// TwinCAT 3 PLC project OC_Core
// Title: OC_Core
// Company: Open Commissioning
// Author: SpiraTec AG
// ProjectVersion: 1.3.1
// Description: Open Commissioning TwinCAT Core Library
// ProgramVersion: 3.1.4026.11
// libraries:
//   Tc2_Math, * (Beckhoff Automation GmbH)
//   Tc2_Standard, * (Beckhoff Automation GmbH)
//   Tc2_System, * (Beckhoff Automation GmbH)
//   Tc2_Utilities, * (Beckhoff Automation GmbH)
//   Tc3_Module, * (Beckhoff Automation GmbH)
//   TcUnit, * (www.tcunit.org)
// project tree:
//   Common/AdsMessageHandler/ FB_AdsMessageHandler.TcPOU, ST_AdsMessage.TcDUT
//   Common/Components/Encoder/ FB_Encoder.TcPOU, ST_Encoder_Config.TcDUT
//   Common/Components/ FB_DriveControl.TcPOU, FB_Clock.TcPOU, FB_ClockAdvanced.TcPOU, FB_Heater.TcPOU, FB_MoveAbsolute.TcPOU, FB_MoveVelocity.TcPOU, FB_Ping.TcPOU
//   Common/FileIo/ E_FileIoState.TcDUT, FB_FileIO.TcPOU
//   Common/Links/ FB_LinkDataReal.TcPOU, FB_LinkDevice.TcPOU, FB_LinkDataWord.TcPOU, FB_LinkDataLWord.TcPOU, FB_LinkDataDWord.TcPOU, FB_LinkDataByte.TcPOU
//   Common/RecordData/ FB_RecordData.TcPOU, I_RecordData.TcIO, ST_RecordIdent.TcDUT
//   Common/System/ E_ControllerType.TcDUT, FB_Base.TcPOU, FB_System.TcPOU, F_LogError.TcPOU, F_LogMessage.TcPOU, F_LogWarning.TcPOU, F_IsSystemValid.TcPOU, GVL_Core.TcGVL
//   Common/Utils/ E_NetworkByteOrder.TcDUT, F_Clamp01.TcPOU, F_GetHByte.TcPOU, F_Compare.TcPOU, F_GetLByte.TcPOU, F_Memcpy.TcPOU, F_Norm.TcPOU, F_ScaleLREAL.TcPOU, F_Sign.TcPOU, F_InverBytesOrder.TcPOU, ST_ScaleConfig.TcDUT
//   Devices/Basic/ FB_Device.TcPOU, FB_Panel.TcPOU, FB_Lock.TcPOU, FB_Cylinder.TcPOU, FB_DeviceByte.TcPOU, FB_DeviceLWord.TcPOU, FB_DeviceWord.TcPOU, FB_DeviceDWord.TcPOU, FB_DeviceReal.TcPOU, FB_Drive.TcPOU, FB_Button.TcPOU, FB_Lamp.TcPOU, FB_Reader.TcPOU, FB_Robot.TcPOU, FB_SensorAnalog.TcPOU, FB_SensorBinary.TcPOU, FB_Switch.TcPOU
//   / PlcTask.TcTTO
//   Tests/Common/ FB_AdsMessageHandler_Test.TcPOU, FB_Encoder_Test.TcPOU, FB_Memcpy_Test.TcPOU, FB_RecordData_Test.TcPOU, FB_Clamp01_Test.TcPOU, FB_Compare_Test.TcPOU, FB_InverBytesOrder_Test.TcPOU, FB_Norm_Test.TcPOU, FB_Sign_Test.TcPOU, FB_Scale_Test.TcPOU, FB_GetByte_Test.TcPOU, FB_System_Test.TcPOU
//   Tests/Components/ FB_DriveControl_Test.TcPOU, FB_Heater_Test.TcPOU, FB_MoveAbsolute_Test.TcPOU, FB_MoveVelocity_Test.TcPOU
//   Tests/Devices/ FB_Button_Test.TcPOU, FB_Device_Test.TcPOU, FB_Switch_Test.TcPOU, FB_Lock_Test.TcPOU, FB_DeviceReal_Test.TcPOU, FB_Panel_Test.TcPOU, FB_Robot_Test.TcPOU, FB_SensorBinary_Test.TcPOU, FB_SensorAnalog_Test.TcPOU, FB_Reader_Test.TcPOU, FB_Lamp_Test.TcPOU, FB_Cylinder_Test.TcPOU, FB_DeviceByte_Test.TcPOU, FB_Drive_Test.TcPOU, FB_DeviceLWord_Test.TcPOU, FB_DeviceWord_Test.TcPOU, FB_DeviceDWord_Test.TcPOU
//   Tests/ PRG_TEST.TcPOU

CONFIGURATION OC_Core
    RESOURCE PLC ON TwinCAT3
        TASK PlcTask(INTERVAL := T#1ms, PRIORITY := 1);
        PROGRAM PRG_TEST WITH PlcTask : PRG_TEST;
    END_RESOURCE
END_CONFIGURATION

// ---- Common/AdsMessageHandler/ST_AdsMessage.TcDUT
TYPE ST_AdsMessage :
STRUCT
	tNetID			: T_AmsNetID; // AMS NetId identifier
	tPort			: T_AmsPort; // AMS port number
	nInvokeID		: UDINT; // Unique identifier for the ADS invocation
	nIdxGrp			: UDINT; // Index group for the ADS command
	nIdxOffs		: UDINT; // Index offset within the ADS command
	nLength			: UDINT; // Length of the ADS message data
	nResult			: UDINT; // Result code from the ADS operation
	aData			: ARRAY[0..239] OF BYTE; // Data payload (240-byte buffer)
END_STRUCT
END_TYPE

// ---- Common/Components/Encoder/ST_Encoder_Config.TcDUT
TYPE ST_Encoder_Config :
STRUCT
	bIsIntegrator   		: BOOL := FALSE;  //Integrate input value
	fNumerator 	  			: REAL := 0.0001; //[unit/INC]
	fDenominator  			: REAL := 1.0; 	// Scaling
	fModulo 	  			: REAL := 0; // Modulo [unit]; If 0, will be ignored
	fGearFactor  			: REAL := 1.0;
	bInvertEncoderDirection : BOOL;
END_STRUCT
END_TYPE

// ---- Common/FileIo/E_FileIoState.TcDUT
{attribute 'conditionalshow'}
TYPE E_FileIoState :
(
	READY := 0,
	OPEN,
	CREATE,
	READ,
	WRITE,
	CLOSE,
	ERROR
);
END_TYPE

// ---- Common/RecordData/ST_RecordIdent.TcDUT
TYPE ST_RecordIdent :
STRUCT
	nPort  			: T_AmsPort; //ADS-Port of the Profinet Device. Ignored when using PLCSIM Advanced
	nSlot			: UINT; //Slotnumber of the Profinet Device. Ignored when using PLCSIM Advanced
	nSubSlot		: UINT; //Subslotnumber of the Profinet Device. Ignored when using PLCSIM Advanced
	nPlcId			: UINT; //Identifier of the PLC when using PLCSIM Advanced
	nHardwareId		: UINT; //Hardware-ID of the device when using PLCSIM Advanced
END_STRUCT
END_TYPE

// ---- Common/System/E_ControllerType.TcDUT
{attribute 'qualified_only'}
{attribute 'strict'}
TYPE E_ControllerType :
(
	NotDefined := 0,
	PlcSimAdvanced := 1
);
END_TYPE

// ---- Common/Utils/E_NetworkByteOrder.TcDUT
{attribute 'qualified_only'}
{attribute 'strict'}
TYPE E_NetworkByteOrder :
(
	BigEndian := 0, //Big Endian (MOTOROLA)
	LittleEndian := 1 //Little Endian (Intel)	
);
END_TYPE

// ---- Common/Utils/ST_ScaleConfig.TcDUT
{attribute 'pack_mode' := '0'} 
TYPE ST_ScaleConfig :
STRUCT
	fInputMin 	: LREAL := 0;
	fInputMax 	: LREAL := 100;
	fOutputMin 	: LREAL := 0;
	fOutputMax 	: LREAL := 65535;
END_STRUCT
END_TYPE

// ---- Common/System/GVL_Core.TcGVL
{attribute 'qualified_only'}
{attribute 'conditionalshow'}
VAR_GLOBAL	
	refSystem 			: REFERENCE TO FB_System;		
END_VAR

// ---- Common/RecordData/I_RecordData.TcIO
{attribute 'conditionalshow'}
INTERFACE I_RecordData

(*Send ADS Read Response message*)
METHOD SendReadResponse : HRESULT
VAR_INPUT
	stAdsMessage : ST_AdsMessage; //Response ADS Message
END_VAR
END_METHOD

(*Send ADS Write Response message*)
METHOD SendWriteResponse : HRESULT
VAR_INPUT
	stAdsMessage : ST_AdsMessage; //Response ADS Message
END_VAR
END_METHOD

(*Try to get a valid ADR read message. If the message is valid, the data in the input structure will be overwritten*)
METHOD GetReadIndication : BOOL
VAR_INPUT
	refDeviceAdsMessage : REFERENCE TO ST_AdsMessage; //Reference ADS Message
END_VAR
END_METHOD

(*Subscribe the RecordIdent device to the RecordData services. The RecordIdent device is initialised during subscription*)
METHOD Subscribe
VAR_INPUT
	pRecordIdent	: POINTER TO ST_RecordIdent; //Pointet to RecordIdent Device
	stAdsMessage 	: REFERENCE TO ST_AdsMessage; //Reference to the initial ADS message configuration of the device
END_VAR
END_METHOD

(*Try to get a valid ADR write message. If the message is valid, the data in the input structure will be overwritten*)
METHOD GetWriteIndication : BOOL
VAR_INPUT
	refDeviceAdsMessage : REFERENCE TO ST_AdsMessage; //Reference ADS Message
END_VAR
END_METHOD

END_INTERFACE

// ---- Tests/PRG_TEST.TcPOU
PROGRAM PRG_TEST
VAR
	FB_System_Test : FB_System_Test;
	FB_Clamp01_Test : FB_Clamp01_Test;
	FB_Compare_Test : FB_Compare_Test;
	FB_Norm_Test : FB_Norm_Test;
	FB_Scale_Test : FB_Scale_Test;
	FB_Sign_Test : FB_Sign_Test;
	FB_InverBytesOrder_Test : FB_InverBytesOrder_Test;
	FB_GetByte_Test : FB_GetByte_Test;
	FB_MEMCPY_Test : FB_MEMCPY_Test;
	FB_Heater_Test : FB_Heater_Test;
	FB_MoveVelocity_Test : FB_MoveVelocity_Test;
	FB_MoveAbsolute_Test : FB_MoveAbsolute_Test; 
	FB_DriveControl_Test : FB_DriveControl_Test;
	FB_Button_Test : FB_Button_Test;
	FB_Switch_Test : FB_Switch_Test;
	FB_Lock_Test : FB_Lock_Test;
	FB_Panel_Test : FB_Panel_Test;
	FB_Cylinder_Test : FB_Cylinder_Test;
	FB_Device_Test : FB_Device_Test;
	FB_DeviceByte_Test : FB_DeviceByte_Test;
	FB_DeviceWord_Test : FB_DeviceWord_Test;
	FB_DeviceDWord_Test : FB_DeviceDWord_Test;
	FB_DeviceLWord_Test : FB_DeviceLWord_Test;
	FB_DeviceReal_Test : FB_DeviceReal_Test;
	FB_Drive_Test : FB_Drive_Test;
	FB_Lamp_Test : FB_Lamp_Test;
	FB_Reader_Test : FB_Reader_Test;
	FB_SensorAnalog_Test : FB_SensorAnalog_Test;
	FB_SensorBinary_Test : FB_SensorBinary_Test;
	FB_Robot_Test : FB_Robot_Test;	
	FB_AdsMessageHandler_Test : FB_AdsMessageHandler_Test;
	FB_RecordData_Test : FB_RecordData_Test;
	FB_Encoder_Test : FB_Encoder_Test;	
END_VAR

TcUnit.RUN();

END_PROGRAM

// ---- Tests/Common/FB_System_Test.TcPOU
FUNCTION_BLOCK FB_System_Test EXTENDS TcUnit.FB_TestSuite
VAR
	_fbSystem : FB_System;
END_VAR

TestInitialization();
TestProperties();

METHOD TestInitialization
VAR
	fbGetCurTaskIdx 	: TC2_SYSTEM.GETCURTASKINDEX;
	fResult 	: REAL;
	fExpected 	: REAL;
	bResult 	: BOOL;
	bExpected 	: BOOL;
END_VAR
TEST('Before InitRun fTimeScaling is 0');
fExpected := 0;
fResult := _fbSystem.fTimeScaling;
AssertEquals(Expected := fExpected,
             Actual := fResult,
             Message := 'Result value is not correct');
TEST_FINISHED();

TEST('Before InitRun fDeltaTime is 0');
fExpected := 0;
fResult := _fbSystem.fDeltaTime;
AssertEquals(Expected := fExpected,
             Actual := fResult,
             Message := 'Result value is not correct');	
TEST_FINISHED();

TEST('Before InitRun GVL_IOSEF.refSystem is NULL');
bExpected := FALSE;
bResult := __ISVALIDREF(GVL_Core.refSystem);
AssertEquals(Expected := bExpected,
             Actual := bResult,
             Message := 'Result value is not correct');	
TEST_FINISHED();

_fbSystem();

TEST('After InitRun fTimeScaling > 0');
fExpected := 1;
fResult := _fbSystem.fTimeScaling;
AssertEquals(Expected := fExpected,
             Actual := fResult,
             Message := 'Result value is not correct');
TEST_FINISHED();

TEST('After InitRun fDeltaTime > 0');
fbGetCurTaskIdx();
fExpected := UDINT_TO_REAL(TwinCAT_SystemInfoVarList._TaskInfo[fbGetCurTaskIdx.index].CycleTime / 10000) / 1000.0;
fResult := _fbSystem.fDeltaTime;
AssertEquals(Expected := fExpected,
             Actual := fResult,
             Message := 'Result value is not correct');	
TEST_FINISHED();

TEST('After InitRun GVL_IOSEF.refSystem is Valid');
bExpected := TRUE;
bResult := __ISVALIDREF(GVL_Core.refSystem);
AssertEquals(Expected := bExpected,
             Actual := bResult,
             Message := 'Result value is not correct');	
TEST_FINISHED();
END_METHOD

METHOD TestProperties : REFERENCE TO FB_Test
VAR
	fbGetCurTaskIdx 	: TC2_SYSTEM.GETCURTASKINDEX;
	fResult 	: REAL;
	fExpected 	: REAL;
END_VAR
TEST('Test Property: bDebug');
_fbSystem.bDebug := TRUE;
AssertTRUE(Condition := _fbSystem.bDebug,  Message := 'Property value is not correct');	
TEST_FINISHED();

TEST('Test Property: bVerbose');
_fbSystem.bVerbose := TRUE;
AssertTRUE(Condition := _fbSystem.bVerbose,  Message := 'Property value is not correct');	
TEST_FINISHED();

TEST('Test Property: fTimeScaling Initial');
fExpected := 1;
fResult := _fbSystem.fTimeScaling;
AssertEquals(Expected := fExpected,
             Actual := fResult,
             Message := 'Result value is not correct');
TEST_FINISHED();

TEST('Test Property: fTimeScaling Zero');
_fbSystem.fTimeScaling := 0;
fExpected := 1;
fResult := _fbSystem.fTimeScaling;
AssertEquals(Expected := fExpected,
             Actual := fResult,
             Message := 'Result value is not correct');
TEST_FINISHED();

TEST('Test Property: fTimeScaling Limit Min');
_fbSystem.fTimeScaling := -1;
fExpected := 0.01000001;
fResult := _fbSystem.fTimeScaling;
AssertEquals(Expected := fExpected,
             Actual := fResult,
             Message := 'Result value is not correct');
TEST_FINISHED();

TEST('Test Property: fTimeScaling Limit Max');
_fbSystem.fTimeScaling := 1E+6;
fExpected := 100;
fResult := _fbSystem.fTimeScaling;
AssertEquals(Expected := fExpected,
             Actual := fResult,
             Message := 'Result value is not correct');
TEST_FINISHED();

TEST('Test Property: fTimeScaling In Range_1');
_fbSystem.fTimeScaling := 2;
fExpected := 2;
fResult := _fbSystem.fTimeScaling;
AssertEquals(Expected := fExpected,
             Actual := fResult,
             Message := 'Result value is not correct');
TEST_FINISHED();

TEST('Test Property: fTimeScaling In Range_2');
_fbSystem.fTimeScaling := 1;
fExpected := 1;
fResult := _fbSystem.fTimeScaling;
AssertEquals(Expected := fExpected,
             Actual := fResult,
             Message := 'Result value is not correct');
TEST_FINISHED();
END_METHOD

END_FUNCTION_BLOCK

// ---- Common/System/FB_System.TcPOU
(*
	FB_System should be defined and called up once in the project so that the GVL reference is correctly assigned. 
	If FB_System is not defined or there are several instances, the TwinCAT PLC project is forced into config mode with corresponding messages in the console.
*)
{attribute 'reflection'} 
FUNCTION_BLOCK FB_System
VAR_INPUT
	fbAdsMessageHandler 	: FB_AdsMessageHandler;
	fbRecordData 			: FB_RecordData(refAdsMessageHandler := fbAdsMessageHandler);
END_VAR

VAR
	{attribute 'simulation_interface'}
	Control				AT %Q* : BYTE;
	{attribute 'simulation_interface'}
	Status				AT %I* : BYTE;
	{attribute 'simulation_interface'}
	TimeScaling			AT %I* : REAL := 1.0;
	
	{attribute 'instance-path'} 
    {attribute 'noinit'} 
	_sPath 				: STRING;
	
	_bDebug				: BOOL;
	_bVerbose			: BOOL;
	_fDeltaTime 		: REAL;
	_fTimeScaling 		: REAL;
	_eControllerType	: E_ControllerType;
	
	_fbPing				: FB_Ping;
	
	{attribute 'hide'}
	_fbGetCurTaskIdx 	: TC2_SYSTEM.GETCURTASKINDEX;
END_VAR

InitRun();
fTimeScaling := TimeScaling;
_fbPing(bFeedback := Status.7, bTrigger => Control.7);

fbRecordData(); //Execution order -1 relative to FB_AdsMessageHandler
fbAdsMessageHandler();

PROPERTY bDebug : BOOL
GET
bDebug := _bDebug;
END_GET
SET
_bDebug := bDebug;
END_SET
END_PROPERTY

PROPERTY bVerbose : BOOL
GET
bVerbose := _bVerbose;
END_GET
SET
_bVerbose := bVerbose;
END_SET
END_PROPERTY

PROPERTY eControllerType : E_ControllerType
GET
eControllerType := _eControllerType;
END_GET
SET
_eControllerType := eControllerType;
END_SET
END_PROPERTY

PROPERTY PUBLIC fDeltaTime : REAL
GET
fDeltaTime := _fDeltaTime;
END_GET
SET // PRIVATE
_fDeltaTime := fDeltaTime;
END_SET
END_PROPERTY

PROPERTY PUBLIC fTimeScaling : REAL
GET
fTimeScaling := _fTimeScaling;
END_GET
SET
IF fTimeScaling = 0 THEN
	_fTimeScaling := 1.0;
ELSE
	_fTimeScaling := LIMIT(0.01000001, fTimeScaling, 100.0);	
END_IF
END_SET
END_PROPERTY

METHOD PRIVATE InitRun
VAR_INST
	bInitRun 			: BOOL := TRUE;
	sMessageFormat   	: T_MAXSTRING := '%s %s';
	sMessage  			: T_MAXSTRING;
	fbFormatString 		: FB_FormatString;
END_VAR
IF NOT bInitRun THEN RETURN; END_IF
bInitRun := FALSE;

IF __ISVALIDREF(GVL_Core.refSystem) THEN	
	fbFormatString(sFormat := sMessageFormat, arg1 := F_STRINGEx(_sPath), arg2 := F_STRINGEx('FB_System has no single instance! Check the PROGRAM declaration'), sOut => sMessage);
	ADSLOGSTR(msgCtrlMask := ADSLOG_MSGTYPE_ERROR, '%s', sMessage);	
ELSE 
	GVL_Core.refSystem REF= THIS^;
END_IF

_fbGetCurTaskIdx();
_fDeltaTime := UDINT_TO_REAL(TwinCAT_SystemInfoVarList._TaskInfo[_fbGetCurTaskIdx.index].CycleTime / 10000) / 1000.0;
_fTimeScaling := 1;

fbRecordData.eControllerType := _eControllerType;
END_METHOD

END_FUNCTION_BLOCK

// ---- Common/AdsMessageHandler/FB_AdsMessageHandler.TcPOU
(*ADS Message Handler is responsible for indication of the ADS Read/Write messages for local NetId and generation of the response message*)
FUNCTION_BLOCK FB_AdsMessageHandler
VAR_INPUT
	bDisable 				: BOOL;	//Deactivate cyclical execution
	bLog					: BOOL;	//Log ADS messages data in the console
	bVerbose				: BOOL; //Log Verbose information in the console
END_VAR

VAR	
	_fbAdsWriteIndicator 	: AdsWriteInd;	
	_fbAdsReadIndicator 	: AdsReadInd;
	_fbAdsWriteResponse		: AdsWriteRes;
	_fbAdsReadResponse		: AdsReadRes;	
	_stAdsMessageWrite		: ST_AdsMessage;
	_stAdsMessageRead		: ST_AdsMessage;
END_VAR

VAR CONSTANT
	S_FORMAT_RECEIVEWRITE	: STRING := 'AdsWriteInd Port: %X, IdxGrp: %X, IdxOffs: %X, InvokeId %X, Length: %X';
	S_FORMAT_RECEIVEREAD	: STRING := 'AdsReadInd Port: %X, IdxGrp: %X, IdxOffs: %X, InvokeId %X, Length: %X';
	S_FORMAT_RESPONSEWRITE	: STRING := 'AdsWriteRes Port: %X, IdxGrp: %X, IdxOffs: %X, InvokeId %X, Length: %X';
	S_FORMAT_RESPONSEREAD	: STRING := 'AdsReadRes Port: %X, IdxGrp: %X, IdxOffs: %X, InvokeId %X, Length: %X';  
END_VAR

IF bDisable THEN RETURN; END_IF

//Reset Indication and Result FBs
_fbAdsWriteResponse(RESPOND := FALSE);
_fbAdsReadResponse(RESPOND := FALSE);

//Capture all Write requests
_fbAdsWriteIndicator();
CreateAdsWriteMessage();
		
//Capture all Read requests
_fbAdsReadIndicator();
CreateAdsReadMessage();

(*Returns the status of the indication of the read message in the current frame*)
PROPERTY PUBLIC bIsAdsMessageReadValid : BOOL
GET
bIsAdsMessageReadValid := _stAdsMessageRead.tPort <> 0;
END_GET
END_PROPERTY

(*Returns the status of the indication of the write message in the current frame*)
PROPERTY PUBLIC bIsAdsMessageWriteValid : BOOL
GET
bIsAdsMessageWriteValid := _stAdsMessageWrite.tPort <> 0;
END_GET
END_PROPERTY

METHOD PRIVATE CreateAdsReadMessage : BOOL
IF NOT _fbAdsReadIndicator.VALID THEN RETURN; END_IF

MEMSET(ADR(_stAdsMessageRead), 0, SIZEOF(ST_AdsMessage));
_stAdsMessageRead.tNetId 		:= _fbAdsReadIndicator.NETID;
_stAdsMessageRead.tPort 		:= _fbAdsReadIndicator.PORT;
_stAdsMessageRead.nInvokeId 	:= _fbAdsReadIndicator.INVOKEID;
_stAdsMessageRead.nIdxGrp 		:= _fbAdsReadIndicator.IDXGRP;
_stAdsMessageRead.nIdxOffs 		:= _fbAdsReadIndicator.IDXOFFS;
_stAdsMessageRead.nLength 		:= _fbAdsReadIndicator.LENGTH;

IF bVerbose THEN
	LogAdsMessage(_stAdsMessageWrite, S_FORMAT_RECEIVEREAD);
END_IF

_fbAdsReadIndicator(CLEAR := TRUE);
_fbAdsReadIndicator(CLEAR := FALSE);
END_METHOD

METHOD PRIVATE CreateAdsWriteMessage : BOOL
IF NOT _fbAdsWriteIndicator.VALID THEN RETURN; END_IF

MEMSET(ADR(_stAdsMessageWrite), 0, SIZEOF(ST_AdsMessage));
_stAdsMessageWrite.tNetId 		:= _fbAdsWriteIndicator.NETID;
_stAdsMessageWrite.tPort 		:= _fbAdsWriteIndicator.PORT;
_stAdsMessageWrite.nInvokeId 	:= _fbAdsWriteIndicator.INVOKEID;
_stAdsMessageWrite.nIdxGrp 		:= _fbAdsWriteIndicator.IDXGRP;
_stAdsMessageWrite.nIdxOffs 	:= _fbAdsWriteIndicator.IDXOFFS;
_stAdsMessageWrite.nLength 		:= _fbAdsWriteIndicator.LENGTH;
			
//Limit size to 240
IF _stAdsMessageWrite.nLength > 240 THEN
	IF bVerbose THEN
		F_LOGWARNING(CONCAT('WRREC data length limited to 240. Requested data length was ', TO_STRING(_stAdsMessageWrite.nLength)));
	END_IF
	_stAdsMessageWrite.nLength := 240;
END_IF

MEMCPY(ADR(_stAdsMessageWrite.aData), _fbAdsWriteIndicator.DATAADDR, _stAdsMessageWrite.nLength);

IF bVerbose THEN
	LogAdsMessage(_stAdsMessageWrite, S_FORMAT_RECEIVEWRITE);
END_IF

_fbAdsWriteIndicator(CLEAR := TRUE);
_fbAdsWriteIndicator(CLEAR := FALSE);
END_METHOD

METHOD PRIVATE LogAdsMessage : BOOL
VAR_INPUT
	stAdsMessage 			: ST_AdsMessage;
	sFormat 				: STRING;
END_VAR

VAR
	fbFormatString			: FB_FormatString2;
	sMessage				: STRING;
END_VAR
fbFormatString(
	pFormatString := ADR(sFormat),
	arg1 := F_UINT(stAdsMessage.tPort),
	arg2 := F_UDINT(stAdsMessage.nIdxGrp),
	arg3 := F_UDINT(stAdsMessage.nIdxOffs),		
	arg4 := F_UDINT(stAdsMessage.nInvokeID),
	arg5 := F_UDINT(stAdsMessage.nLength),
	pDstString := ADR(sMessage),
	nDstSize := SIZEOF(sMessage));
F_LogMessage(sMessage);
END_METHOD

(*Send ADS Read Response message*)
METHOD PUBLIC SendReadResponse : HRESULT
VAR_INPUT
	stAdsMessage 	: ST_AdsMessage; //Response ADS Message
END_VAR
IF _fbAdsReadResponse.RESPOND THEN
	SendReadResponse := S_PENDING;
	RETURN;
END_IF

//Limit size to 240
IF stAdsMessage.nLength > 240 THEN
	IF bVerbose THEN
		F_LOGWARNING(CONCAT('RDRES data length limited to 240. Requested data length was ', TO_STRING(stAdsMessage.nLength)));
	END_IF
	stAdsMessage.nLength := 240;
END_IF

_fbAdsReadResponse(
	NETID:= stAdsMessage.tNetId, 
	PORT:= stAdsMessage.tPort, 
	INVOKEID:= stAdsMessage.nInvokeId, 
	RESULT:= stAdsMessage.nResult, 
	LEN:= stAdsMessage.nLength,
	DATAADDR:= ADR(stAdsMessage.aData),
	RESPOND:= TRUE);
IF bVerbose OR bLog THEN	
	LogAdsMessage(stAdsMessage, S_FORMAT_RESPONSEREAD);
END_IF

SendReadResponse := S_OK;
END_METHOD

(*Send ADS Write Response message*)
METHOD PUBLIC SendWriteResponse : HRESULT
VAR_INPUT
	stAdsMessage 	: ST_AdsMessage; //Response ADS Message
END_VAR
IF _fbAdsWriteResponse.RESPOND THEN
	SendWriteResponse := S_PENDING;
	RETURN;
END_IF

_fbAdsWriteResponse(
	NETID:= stAdsMessage.tNetId, 
	PORT:= stAdsMessage.tPort, 
	INVOKEID:= stAdsMessage.nInvokeId, 
	RESULT:= stAdsMessage.nResult, 
	RESPOND:= TRUE);	

IF bVerbose OR bLog THEN		
	LogAdsMessage(stAdsMessage, S_FORMAT_RESPONSEWRITE);
END_IF
	
SendWriteResponse := S_OK;
END_METHOD

(*Get last valid ADS Read Message*)
PROPERTY stAdsMessageRead : REFERENCE TO ST_AdsMessage
GET
stAdsMessageRead REF= _stAdsMessageRead;
END_GET
END_PROPERTY

(*Get last valid ADS Write Message*)
PROPERTY stAdsMessageWrite : REFERENCE TO ST_AdsMessage
GET
stAdsMessageWrite REF= _stAdsMessageWrite;
END_GET
END_PROPERTY

END_FUNCTION_BLOCK

// ---- Common/System/F_LogWarning.TcPOU
(*
	Log Warning message to TwinCAT console
*)
{attribute 'hide_all_locals'}
FUNCTION F_LogWarning : BOOL
VAR_INPUT
	sMessage : T_MAXSTRING;
END_VAR

VAR CONSTANT	
	S_LOGHEADER		: T_MAXSTRING := 'Open Commissioning: %s';
END_VAR

ADSLOGSTR(ADSLOG_MSGTYPE_WARN, S_LOGHEADER, sMessage);

END_FUNCTION

// ---- Common/System/F_LogMessage.TcPOU
(*
	Log message to TwinCAT console
*)
{attribute 'hide_all_locals'}
FUNCTION F_LogMessage : BOOL
VAR_INPUT
	sMessage : T_MAXSTRING;
END_VAR

VAR CONSTANT	
	S_LOGHEADER		: T_MAXSTRING := 'Open Commissioning: %s';
END_VAR

ADSLOGSTR(ADSLOG_MSGTYPE_HINT, S_LOGHEADER, sMessage);

END_FUNCTION

// ---- Common/RecordData/FB_RecordData.TcPOU
(*
	Uses an external ADS message handler (FB_AdsMessageHandler) for sending/receiving ADS messages.
	Handles cyclic execution for processing ADS messages and maintains a list of subscribed devices.	
*)
{attribute 'conditionalshow_all_locals}
FUNCTION_BLOCK PUBLIC FB_RecordData IMPLEMENTS I_RecordData
VAR_INPUT
	bDisable 				: BOOL; //Disables cyclic execution when set to TRUE
	bVerbose 				: BOOL; //Enables console logging of ADS message data
	eControllerType 		: E_ControllerType; //Determines data processing logic based on the controller type
END_VAR

VAR	
	_refAdsMessageHandler	: REFERENCE TO FB_AdsMessageHandler;	//Reference to the external ADS message handler used for managing ADS messages	
	_nDeviceCount			: INT;	//Number of devices subscribed for record data
	_aDeviceList			: ARRAY[0..255] OF UDINT; //The internal device list is used for assistance services. Do not delete or change. 
END_VAR

IF bDisable THEN RETURN; END_IF

//Send WriteRes if last WriteInd has not been read by any device
IF _refAdsMessageHandler.stAdsMessageWrite.tPort <> 0 THEN
	SendWriteResponse(_refAdsMessageHandler.stAdsMessageRead);
	_refAdsMessageHandler.stAdsMessageWrite.tPort := 0;
END_IF

//Send ReadRes if last ReadInd has not been read by any device
IF _refAdsMessageHandler.stAdsMessageRead.tPort <> 0 THEN
	SendReadResponse(_refAdsMessageHandler.stAdsMessageRead);
	_refAdsMessageHandler.stAdsMessageRead.tPort := 0;
END_IF 

(*Ads Message Comments*)
//tNetId			: T_AmsNetID;
//tPort				: T_AmsPort;
//nInvokeId			: UDINT; //Hil: Byte0 and 1 = Port, Byte2 = Subslot, Byte3 = Slot. Sil: ignored.
//nIndexGroup		: UDINT; //16#80000000 + RecordIndex
//nIndexOffset		: UDINT; //Hil: LowWord = SubSlot, HighWord = Slot. Sil: LowWord = HardwareId, HighWord = PlcId.
//nLengthData		: UDINT;
//nResult			: UDINT;
//aData				: ARRAY[0..239] OF BYTE;

METHOD PRIVATE CmpIGrp : BOOL
VAR_INPUT
	nIGrpDevice 	: UDINT;
	nIGrpReceived 	: UDINT;
END_VAR
(* Compare low word only *)
CmpIGrp := (nIGrpDevice AND 16#0000FFFF) = (nIGrpReceived AND 16#0000FFFF) OR nIGrpDevice = 0;
END_METHOD

METHOD PRIVATE CmpInvokeId : BOOL
VAR_INPUT
	nInvokeIdDevice 	: UDINT;
	nInvokeIdReceived 	: UDINT;
END_VAR
IF eControllerType = E_ControllerType.PlcSimAdvanced THEN
	CmpInvokeId := TRUE;
	RETURN;
END_IF

(* Compare low word only. low word = port *)
CmpInvokeId := (nInvokeIdDevice AND 16#0000FFFF) = (nInvokeIdReceived AND 16#0000FFFF);
END_METHOD

METHOD PRIVATE CmpIOffs : BOOL
VAR_INPUT
	nIOffsDevice 	: UDINT;
	nIOffsReceived 	: UDINT;
END_VAR
CmpIOffs := nIOffsDevice = nIOffsReceived OR nIOffsDevice = 16#FFFFFFFF;
END_METHOD

METHOD INTERNAL DataValid : BOOL
VAR_INPUT
	refDeviceAdsMessage 	: REFERENCE TO ST_AdsMessage;
	refHandlerAdsMessage	: REFERENCE TO ST_AdsMessage;
END_VAR
DataValid := FALSE;

IF refHandlerAdsMessage.tPort = 0 THEN
	RETURN;
END_IF

IF NOT CmpInvokeId(refDeviceAdsMessage.nInvokeId, refHandlerAdsMessage.nInvokeId) THEN
	RETURN;
END_IF

IF NOT CmpIOffs(refDeviceAdsMessage.nIdxOffs, refHandlerAdsMessage.nIdxOffs) THEN
	RETURN;
END_IF

IF NOT CmpIGrp(refDeviceAdsMessage.nIdxGrp, refHandlerAdsMessage.nIdxGrp) THEN
	RETURN;
END_IF

(* Copy the received telegram *)
MEMCPY(ADR(refDeviceAdsMessage), ADR(refHandlerAdsMessage), SIZEOF(ST_AdsMessage));

(* Indicate that the telegram has been read by a device
   -> the device is now responsible for the response! *)
refHandlerAdsMessage.tPort := 0;

DataValid := TRUE;
END_METHOD

METHOD FB_init : BOOL
VAR_INPUT
	bInitRetains 				: BOOL; // if TRUE, the retain variables are initialized (warm start / cold start)
	bInCopyCode 				: BOOL;  // if TRUE, the instance afterwards gets moved into the copy code (online change)
	refAdsMessageHandler		: REFERENCE TO FB_AdsMessageHandler;
END_VAR
THIS^._refAdsMessageHandler REF= refAdsMessageHandler;
END_METHOD

(*Try to get a valid ADR read message. If the message is valid, the data in the input structure will be overwritten*)
METHOD PUBLIC GetReadIndication : BOOL
VAR_INPUT
	refDeviceAdsMessage : REFERENCE TO ST_AdsMessage; //Reference ADS Message
END_VAR
IF NOT _refAdsMessageHandler.bIsAdsMessageReadValid THEN
	GetReadIndication := FALSE;
	RETURN; 
END_IF

GetReadIndication := DataValid(refDeviceAdsMessage, _refAdsMessageHandler.stAdsMessageRead);
END_METHOD

(*Try to get a valid ADR write message. If the message is valid, the data in the input structure will be overwritten*)
METHOD PUBLIC GetWriteIndication : BOOL
VAR_INPUT
	refDeviceAdsMessage : REFERENCE TO ST_AdsMessage; //Reference ADS Message	
END_VAR
IF NOT _refAdsMessageHandler.bIsAdsMessageWriteValid THEN
	GetWriteIndication := FALSE;
	RETURN; 
END_IF

GetWriteIndication := DataValid(refDeviceAdsMessage, _refAdsMessageHandler.stAdsMessageWrite);
END_METHOD

(*Send ADS Read Response message*)
METHOD PUBLIC SendReadResponse : HRESULT
VAR_INPUT
	stAdsMessage : ST_AdsMessage; //Response ADS Message
END_VAR
CASE eControllerType OF		
	E_ControllerType.PlcSimAdvanced :
		stAdsMessage.nResult := SHR(stAdsMessage.nIdxOffs, 16) + 16#80000000;
END_CASE

SendReadResponse := _refAdsMessageHandler.SendReadResponse(stAdsMessage);
END_METHOD

(*Send ADS Write Response message*)
METHOD PUBLIC SendWriteResponse : HRESULT
VAR_INPUT
	stAdsMessage : ST_AdsMessage; //Response ADS Message
END_VAR
CASE eControllerType OF		
	E_ControllerType.PlcSimAdvanced :
		stAdsMessage.nResult := SHR(stAdsMessage.nIdxOffs, 16) + 16#80000000;
END_CASE

SendWriteResponse := _refAdsMessageHandler.SendWriteResponse(stAdsMessage);
END_METHOD

(*Subscribe the RecordIdent device to the RecordData services. The RecordIdent device is initialised during subscription*)
METHOD PUBLIC Subscribe
VAR_INPUT
	pRecordIdent	: POINTER TO ST_RecordIdent; //Pointet to RecordIdent Device
	stAdsMessage 	: REFERENCE TO ST_AdsMessage; //Reference to the initial ADS message configuration of the device
END_VAR
IF _nDeviceCount > 255 THEN
	F_LogError('More than 256 RecordData devices');
	RETURN;
END_IF

CASE eControllerType OF
	E_ControllerType.NotDefined :	
		stAdsMessage.nInvokeId := pRecordIdent^.nPort + UINT_TO_USINT(pRecordIdent^.nSubSlot) * 16#10000 + UINT_TO_USINT(pRecordIdent^.nSlot) * 16#1000000;		
		stAdsMessage.nIdxOffs := pRecordIdent^.nSubSlot + pRecordIdent^.nSlot * 16#10000;	
		stAdsMessage.tPort := pRecordIdent^.nPort;
		
		IF stAdsMessage.nInvokeId = 0 THEN
			RETURN;
		END_IF
		
		_aDeviceList[_nDeviceCount] := stAdsMessage.nInvokeId;
	
	E_ControllerType.PlcSimAdvanced :
		stAdsMessage.nIdxOffs := pRecordIdent^.nHardwareId + pRecordIdent^.nPlcId * 16#10000;
		
		IF stAdsMessage.nIdxOffs = 0 THEN
			RETURN;
		END_IF
		
		_aDeviceList[_nDeviceCount] := stAdsMessage.nIdxOffs;
END_CASE	

_nDeviceCount := _nDeviceCount + 1;
END_METHOD

END_FUNCTION_BLOCK

// ---- Common/System/F_LogError.TcPOU
(*
	Log Error message to TwinCAT console
*)
{attribute 'hide_all_locals'}
FUNCTION F_LogError : BOOL
VAR_INPUT
	sMessage : T_MAXSTRING;
END_VAR

VAR CONSTANT	
	S_LOGHEADER		: T_MAXSTRING := 'Open Commissioning: %s';
END_VAR

ADSLOGSTR(ADSLOG_MSGTYPE_ERROR, S_LOGHEADER, sMessage);

END_FUNCTION

// ---- Common/Components/FB_Ping.TcPOU
(*
	FB for measuring the delay between trigger and feeback signal
	Already in use for measuring the delay between TwinCAT and Unity components
*)

FUNCTION_BLOCK FB_Ping
VAR_INPUT	
	bFeedback 		: BOOL;	// bit from unity status
END_VAR

VAR_OUTPUT
	bTrigger		: BOOL;	// bit to unity control
	nActET			: DWORD;	// elapsed time in ms
	nMaxET			: DWORD;	// max. elapsed time in ms
END_VAR

VAR	
	_bEnable			: BOOL;
	_fbTrigStart		: R_TRIG;
	_fbTrigStop			: R_TRIG;
	_fbTrigRestart 		: F_TRIG;
	_nTimeStart 		: TIME;
	_nTimeStop 			: TIME;
END_VAR

InitRun();

_fbTrigStart(CLK := _bEnable);
_fbTrigStop(CLK := bFeedback);
_fbTrigRestart(CLK := bFeedback);

IF _fbTrigStart.Q OR _fbTrigRestart.Q THEN
	nActET := 0;
	bTrigger := TRUE;
	_nTimeStart := TIME();
END_IF


IF _fbTrigStop.Q THEN
	bTrigger := FALSE;
	_nTimeStop := TIME();
	nActET := TIME_TO_DWORD(_nTimeStop - _nTimeStart);
	IF nActET >= nMaxET THEN
		nMaxET := nActET;
	END_IF
END_IF

METHOD INTERNAL InitRun
VAR_INST
	bInitRun : BOOL := TRUE;
END_VAR
IF NOT bInitRun THEN RETURN; END_IF

bInitRun := FALSE;
nActET := 0;
nMaxET := 0;
END_METHOD

END_FUNCTION_BLOCK

// ---- Tests/Common/FB_Clamp01_Test.TcPOU
FUNCTION_BLOCK FB_Clamp01_Test EXTENDS TcUnit.FB_TestSuite

TestCase('Value Limit Min Overflow', fValue := -0.1, fExpected:= 0);
TestCase('Value Limit Min',fValue := 0.0, fExpected:= 0);
TestCase('Value In Range ',fValue := 0.5, fExpected:= 0.5);
TestCase('Value Limit Max',fValue := 1, fExpected:= 1);
TestCase('Value Limit Max Overflow',fValue := 1.1, fExpected:= 1);

METHOD TestCase
VAR_INPUT
	sName : T_MaxString;
	fValue : REAL;
	fExpected : REAL;
END_VAR

VAR	
	fResult : REAL;
END_VAR
TEST(sName);
	
fResult := F_Clamp01(fValue);
AssertEquals(Expected := fExpected,
             Actual := fResult,
             Message := 'Result value is not correct');	
	 
TEST_FINISHED();
END_METHOD

END_FUNCTION_BLOCK

// ---- Common/Utils/F_Clamp01.TcPOU
(*
	Clamp the input value within the range of 0 to 1
*)
FUNCTION F_Clamp01 : REAL
VAR_INPUT
	fValue : REAL;
END_VAR

F_Clamp01:= LIMIT(0, fValue, 1);

END_FUNCTION

// ---- Tests/Common/FB_Compare_Test.TcPOU
FUNCTION_BLOCK FB_Compare_Test EXTENDS TcUnit.FB_TestSuite

TestCase('Compare Valid_1', fValueA := 0.0, fValueB := 0.0, fTolerance := 1E-6, bExpected:= TRUE);
TestCase('Compare Valid_2', fValueA := -1E-6, fValueB := -1E-6, fTolerance := 1E-6, bExpected:= TRUE);
TestCase('Compare Valid_3', fValueA := 1E-6, fValueB := 1E-6, fTolerance := 1E-6, bExpected:= TRUE);

TestCase('Compare Not Valid_1', fValueA := 0.0, fValueB := 0.00001, fTolerance := 1E-6, bExpected:= FALSE);
TestCase('Compare Not Valid_2', fValueA := -10, fValueB := -10.00001, fTolerance := 1E-6, bExpected:= FALSE);
TestCase('Compare Not Valid_3', fValueA := 100, fValueB := 100.00001, fTolerance := 1E-6, bExpected:= FALSE);

TestCase('Compare InRange_1', fValueA := 0.0, fValueB := 4.99999, fTolerance := 5, bExpected:= TRUE);
TestCase('Compare InRange_2', fValueA := -1, fValueB := -5.99999, fTolerance := 5, bExpected:= TRUE);
TestCase('Compare InRange_3', fValueA := 1, fValueB := 5.99999, fTolerance := 5, bExpected:= TRUE);

TestCase('Compare Not InRange_1', fValueA := 0.0, fValueB := 5.00000, fTolerance := 5, bExpected:= FALSE);
TestCase('Compare Not InRange_2', fValueA := -1, fValueB := -6.00000, fTolerance := 5, bExpected:= FALSE);
TestCase('Compare Not InRange_3', fValueA := 1, fValueB := 6.00000, fTolerance := 5, bExpected:= FALSE);

METHOD TestCase
VAR_INPUT
	sName : T_MaxString;
	fValueA : REAL;
	fValueB : REAL;
	fTolerance : REAL; 
	bExpected : BOOL;
END_VAR

VAR	
	bResult : BOOL;
END_VAR
TEST(sName);
	
bResult := F_Compare(fValueA, fValueB, fTolerance);
AssertEquals(Expected := bExpected,
             Actual := bResult,
             Message := 'Result value is not correct');	
	 
TEST_FINISHED();
END_METHOD

END_FUNCTION_BLOCK

// ---- Common/Utils/F_Compare.TcPOU
(*
	Compare fValueA and fValueB within the specified fTolerance window
*)
{attribute 'hide_all_locals'}
FUNCTION F_Compare : BOOL
VAR_INPUT
	fValueA 		: REAL;
	fValueB 		: REAL;
	fTolerance 		: REAL := 1E-6;	
END_VAR

VAR
	_fDifference 	: REAL;
END_VAR

_fDifference := ABS(fValueB - fValueA);
fTolerance := LIMIT(1E-6, ABS(fTolerance), 1E+6);
F_Compare := fTolerance > _fDifference;

END_FUNCTION

// ---- Tests/Common/FB_Norm_Test.TcPOU
FUNCTION_BLOCK FB_Norm_Test EXTENDS TcUnit.FB_TestSuite

TestCase('Normalize in Range_1', fMin := 0.0, fMax := 100, fValue := 0, fExpected:= 0);
TestCase('Normalize in Range_2', fMin := 0.0, fMax := 100, fValue := 20, fExpected:= 0.2);
TestCase('Normalize in Range_3', fMin := 0.0, fMax := 100, fValue := 70, fExpected:= 0.7);
TestCase('Normalize in Range_4', fMin := 0.0, fMax := 100, fValue := 100, fExpected:= 1);
TestCase('Normalize in Range_5', fMin := -100, fMax := 100, fValue := 0, fExpected:= 0.5);

TestCase('Normalize Overflow_1', fMin := -100, fMax := 100, fValue := -101, fExpected:= 0);
TestCase('Normalize Overflow_2', fMin := -100, fMax := 100, fValue := 101, fExpected:= 1);

METHOD TestCase
VAR_INPUT
	sName : T_MaxString;
	fMin : REAL;
	fMax : REAL;
	fValue : REAL; 
	fExpected : REAL;
END_VAR

VAR	
	fResult : REAL;
END_VAR
TEST(sName);
	
fResult := F_Norm(fMin, fMax, fValue);
AssertEquals(Expected := fExpected,
             Actual := fResult,
             Message := 'Result value is not correct');	
	 
TEST_FINISHED();
END_METHOD

END_FUNCTION_BLOCK

// ---- Common/Utils/F_Norm.TcPOU
(*
	The input value will be normalized in the range of fMin to fMax.
	The returned value is within the range of 0 to 1.
*)
FUNCTION F_Norm : REAL
VAR_INPUT
	fMin 		: REAL; //Limit Min
	fMax 		: REAL; //Limit Max
	fValue 		: REAL; //Input Value
END_VAR

F_Norm := F_Clamp01((fValue - fMin)/(fMax - fMin));

END_FUNCTION

// ---- Tests/Common/FB_Scale_Test.TcPOU
FUNCTION_BLOCK FB_Scale_Test EXTENDS TcUnit.FB_TestSuite

TestCase('Scale InRange_1', 
fInputMin := 0.0, fInputMax := 100, 
fOutputMin := 0, fOutputMax:= 1000, 
fValue := 0, fExpected:= 0);

TestCase('Scale InRange_2', 
fInputMin := 0.0, fInputMax := 100, 
fOutputMin := 0, fOutputMax:= 1000, 
fValue := 50, fExpected:= 500);

TestCase('Scale InRange_3', 
fInputMin := 0.0, fInputMax := 100, 
fOutputMin := 0, fOutputMax:= 1000, 
fValue := 100, fExpected:= 1000);

TestCase('Scale Overflow_1', 
fInputMin := 0.0, fInputMax := 100, 
fOutputMin := 0, fOutputMax:= 1000, 
fValue := -100, fExpected:= 0);

TestCase('Scale Overflow_2', 
fInputMin := 0.0, fInputMax := 100, 
fOutputMin := 0, fOutputMax:= 1000, 
fValue := 200, fExpected:= 1000);

TestInputValidation('Inputs Valid_1', 
fInputMin := 0.0, fInputMax := 100, 
fOutputMin := 0, fOutputMax:= 1000, bExpected:= FALSE);

TestInputValidation('Inputs Valid_2', 
fInputMin := 99.99, fInputMax := 100, 
fOutputMin := 999.99, fOutputMax:= 1000, bExpected:= FALSE);

TestInputValidation('Inputs Not Valid_1', 
fInputMin := 100, fInputMax := 100, 
fOutputMin := 0, fOutputMax:= 1000, bExpected:= TRUE);

TestInputValidation('Inputs Not Valid_2', 
fInputMin := 100.0001, fInputMax := 100, 
fOutputMin := 0, fOutputMax:= 1000, bExpected:= TRUE);

TestInputValidation('Inputs Not Valid_3', 
fInputMin := 0, fInputMax := 100, 
fOutputMin := 1000, fOutputMax:= 1000, bExpected:= TRUE);

TestInputValidation('Inputs Not Valid_4', 
fInputMin := 0, fInputMax := 100, 
fOutputMin := 1000.001, fOutputMax:= 1000, bExpected:= TRUE);

METHOD TestCase
VAR_INPUT
	sName : T_MaxString;	
	fInputMin 	: LREAL;
	fInputMax 	: LREAL;
	fOutputMin 	: LREAL;
	fOutputMax 	: LREAL;
	fValue 		: LREAL; 
	fExpected 	: LREAL;
END_VAR

VAR	
	fResult 	: LREAL;
END_VAR
TEST(sName);
	
fResult := F_ScaleLREAL(fValue, fInputMin, fInputMax, fOutputMin, fOutputMax);
AssertEquals(Expected := fExpected,
             Actual := fResult,
             Message := 'Result value is not correct');	
	 
TEST_FINISHED();
END_METHOD

METHOD TestInputValidation : REFERENCE TO FB_Test
VAR_INPUT
	sName : T_MaxString;	
	fInputMin 	: LREAL;
	fInputMax 	: LREAL;
	fOutputMin 	: LREAL;
	fOutputMax 	: LREAL;
	bExpected 	: BOOL;
END_VAR

VAR	
	bResult 	: BOOL;
END_VAR
TEST(sName);
	
F_ScaleLREAL(0, fInputMin, fInputMax, fOutputMin, fOutputMax, bError => bResult);
AssertEquals(Expected := bExpected,
             Actual := bResult,
             Message := 'Result value is not correct');	
	 
TEST_FINISHED();
END_METHOD

END_FUNCTION_BLOCK

// ---- Common/Utils/F_ScaleLREAL.TcPOU
(*
 	The input value will be normalize scaled from the input range [fInputMin..fInputMax] to the output range [fOutputMin..fOutputMax].	
*)
FUNCTION F_ScaleLREAL : LREAL
VAR_INPUT
	fValue 		: LREAL; //Input value
	fInputMin 	: LREAL; //Input limit Min
	fInputMax 	: LREAL; //Input limit Max
	fOutputMin 	: LREAL; //Output limit Min
	fOutputMax 	: LREAL; //Output limit Max
END_VAR

VAR
	fNormalized : LREAL;
END_VAR

VAR_OUTPUT
	bError 		: BOOL;
END_VAR

bError := (fInputMin >= fInputMax) OR (fOutputMin >= fOutputMax);

IF bError THEN
	F_ScaleLREAL := 0.0;
	RETURN;
END_IF

IF fValue < fInputMin THEN
	fNormalized := 0.0;
ELSIF fValue > fInputMax THEN
	fNormalized := 1.0;
ELSE
	fNormalized := (fValue - fInputMin) / (fInputMax - fInputMin);
END_IF

F_ScaleLREAL := fNormalized * (fOutputMax - fOutputMin) + fOutputMin;

END_FUNCTION

// ---- Tests/Common/FB_Sign_Test.TcPOU
FUNCTION_BLOCK FB_Sign_Test EXTENDS TcUnit.FB_TestSuite

TestCase('Sign Negative_1', fValue := -0.00001, fExpected:= -1);
TestCase('Sign Negative_2', fValue := -0.1, fExpected:= -1);
TestCase('Sign Negative_3', fValue := -1, fExpected:= -1);

TestCase('Sign Positive_1', fValue := 0, fExpected:= 1);
TestCase('Sign Positive_2', fValue := 0.00001, fExpected:= 1);
TestCase('Sign Positive_3', fValue := 0.1, fExpected:= 1);
TestCase('Sign Positive_4', fValue := 1, fExpected:= 1);

METHOD TestCase
VAR_INPUT
	sName : T_MaxString;	
	fValue : REAL; 
	fExpected : REAL;
END_VAR

VAR	
	fResult : REAL;
END_VAR
TEST(sName);
	
fResult := F_Sign(fValue);
AssertEquals(Expected := fExpected,
             Actual := fResult,
             Message := 'Result value is not correct');	
	 
TEST_FINISHED();
END_METHOD

END_FUNCTION_BLOCK

// ---- Common/Utils/F_Sign.TcPOU
(*
	Return sign of input value
*)
{attribute 'hide_all_locals'}
FUNCTION F_Sign : REAL
VAR_INPUT
	fValue 	: REAL;
END_VAR

IF (fValue >= 0) THEN
	F_Sign := 1;
ELSE
	F_Sign := -1;	
END_IF

END_FUNCTION

// ---- Tests/Common/FB_InverBytesOrder_Test.TcPOU
FUNCTION_BLOCK FB_InverBytesOrder_Test EXTENDS TcUnit.FB_TestSuite

TestWord('Invert WORD_1', nData := 16#1234, nExpected:= 16#3412);
TestWord('Invert WORD_2', nData := 16#4321, nExpected:= 16#2143);

TestDWord('Invert DWORD_1', nData := 16#12345678, nExpected:= 16#78563412);
TestDWord('Invert DWORD_2', nData := 16#87654321, nExpected:= 16#21436587);

TestLWord('Invert LWORD_1', nData := 16#1234567812345678, nExpected:= 16#7856341278563412);
TestLWord('Invert LWORD_2', nData := 16#8765432187654321, nExpected:= 16#2143658721436587);

METHOD TestDWord
VAR_INPUT
	sName : T_MaxString;	
	nData 	: DWORD;
	nExpected : DWORD;
END_VAR

VAR		
	nResult : DWORD;
END_VAR
TEST(sName);


F_InverBytesOrder(nData);
AssertEquals(Expected := nExpected,
             Actual := nData,
             Message := 'Result value is not correct');	
	 
TEST_FINISHED();
END_METHOD

METHOD TestLWord
VAR_INPUT
	sName : T_MaxString;	
	nData 	: LWORD;
	nExpected : LWORD;
END_VAR

VAR		
	nResult : LWORD;
END_VAR
TEST(sName);


F_InverBytesOrder(nData);
AssertEquals(Expected := nExpected,
             Actual := nData,
             Message := 'Result value is not correct');	
	 
TEST_FINISHED();
END_METHOD

METHOD TestWord
VAR_INPUT
	sName : T_MaxString;	
	nData 	: WORD;
	nExpected : WORD;
END_VAR

VAR		
	nResult : WORD;
END_VAR
TEST(sName);


F_InverBytesOrder(nData);
AssertEquals(Expected := nExpected,
             Actual := nData,
             Message := 'Result value is not correct');	
	 
TEST_FINISHED();
END_METHOD

END_FUNCTION_BLOCK

// ---- Common/Utils/F_InverBytesOrder.TcPOU
(*
	Reverse the byte order of the given ANY input.
*)
FUNCTION F_InverBytesOrder : BOOL
VAR_INPUT
	data 	: ANY;
END_VAR

VAR	
	_i 		: UDINT;
	_nSize	: UDINT;
	_aData 	: ARRAY [0..7] OF BYTE;
END_VAR

_nSize := DINT_TO_UDINT(data.diSize);
MEMCPY(ADR(_aData), data.pValue, _nSize);

IF(_nSize > 8) THEN
	F_LogError('F_InverBytesOrder: Data Size is not in range [0..7]');
	RETURN;
END_IF

FOR _i:= 1 TO _nSize DO	
	MEMCPY(data.pValue + _i - 1, ADR(_aData) + _nSize - _i, 1);
END_FOR

END_FUNCTION

// ---- Tests/Common/FB_GetByte_Test.TcPOU
FUNCTION_BLOCK FB_GetByte_Test EXTENDS TcUnit.FB_TestSuite

TestGetLByte('Get LByte_1', nData := 16#1234, nExpected:= 16#34);
TestGetLByte('Get LByte_2', nData := 16#4321, nExpected:= 16#21);

TestGetHByte('Get HByte_1', nData := 16#1234, nExpected:= 16#12);
TestGetHByte('Get HByte_2', nData := 16#4321, nExpected:= 16#43);

METHOD TestGetHByte
VAR_INPUT
	sName : T_MaxString;	
	nData 	: WORD;
	nExpected : BYTE;
END_VAR

VAR		
	nResult : BYTE;
END_VAR
TEST(sName);


nResult := F_GetHByte(nData);
AssertEquals(Expected := nExpected,
             Actual := nResult,
             Message := 'Result value is not correct');	
	 
TEST_FINISHED();
END_METHOD

METHOD TestGetLByte
VAR_INPUT
	sName : T_MaxString;	
	nData 	: WORD;
	nExpected : BYTE;
END_VAR

VAR		
	nResult : BYTE;
END_VAR
TEST(sName);


nResult := F_GetLByte(nData);
AssertEquals(Expected := nExpected,
             Actual := nResult,
             Message := 'Result value is not correct');	
	 
TEST_FINISHED();
END_METHOD

END_FUNCTION_BLOCK

// ---- Common/Utils/F_GetHByte.TcPOU
(*
	Return the high byte from the input word
*)
FUNCTION F_GetHByte : BYTE
VAR_INPUT
	nWord	: WORD;
END_VAR

F_GetHByte := WORD_TO_BYTE(SHR(nWord, 8));

END_FUNCTION

// ---- Common/Utils/F_GetLByte.TcPOU
(*
	Return the low byte from the input word
*)
FUNCTION F_GetLByte : BYTE
VAR_INPUT
	nWord	: WORD;
END_VAR

F_GetLByte := WORD_TO_BYTE(nWord);

END_FUNCTION

// ---- Tests/Common/FB_Memcpy_Test.TcPOU
FUNCTION_BLOCK FB_Memcpy_Test EXTENDS TcUnit.FB_TestSuite

TestCaseWORD();
TestCaseDWORD();
TestCaseLWORD();

METHOD TestCaseDWORD
VAR	
	nValue 				: DWORD;
	nValueExpected 		: DWORD;
	nValueActual 		: DWORD;
END_VAR
TEST('MEMCPY DWORD');
	
//Arrange
nValue := nValueExpected := 16#A1B2C3D4;

//Act
F_MEMCPY(ADR(nValueActual), ADR(nValue), 4, FALSE);

//Assert
AssertEquals(Expected := nValueExpected,
             Actual := nValueActual,
             Message := 'nValueActual not returning expected value');
	 
TEST_FINISHED();


TEST('MEMCPY DWORD SWAP');
	
//Arrange
nValue := 16#A1B2C3D4;
nValueExpected := HOST_TO_BE32(nValue);

//Act
F_MEMCPY(ADR(nValueActual), ADR(nValue), 4, TRUE);

//Assert
AssertEquals(Expected := nValueExpected,
             Actual := nValueActual,
             Message := 'nValueActual not returning expected value');
	 
TEST_FINISHED();
END_METHOD

METHOD TestCaseLWORD
VAR	
	nValue 				: LWORD;
	nValueExpected 		: LWORD;
	nValueActual 		: LWORD;
END_VAR
TEST('MEMCPY LDWORD');
	
//Arrange
nValue := nValueExpected := 16#A1B2C3D4F5E6F701;

//Act
F_MEMCPY(ADR(nValueActual), ADR(nValue), 8, FALSE);

//Assert
AssertEquals(Expected := nValueExpected,
             Actual := nValueActual,
             Message := 'nValueActual not returning expected value');
	 
TEST_FINISHED();


TEST('MEMCPY LDWORD SWAP');
	
//Arrange
nValue := 16#A1B2C3D4F5E6F701;
nValueExpected := HOST_TO_BE64EX(nValue);

//Act
F_MEMCPY(ADR(nValueActual), ADR(nValue), 8, TRUE);

//Assert
AssertEquals(Expected := nValueExpected,
             Actual := nValueActual,
             Message := 'nValueActual not returning expected value');
	 
TEST_FINISHED();
END_METHOD

METHOD TestCaseWORD
VAR	
	nValue 				: WORD;
	nValueExpected 		: WORD;
	nValueActual 		: WORD;
END_VAR
TEST('MEMCPY WORD');
	
//Arrange
nValue := nValueExpected := 16#A1B2;

//Act
F_MEMCPY(ADR(nValueActual), ADR(nValue), 2, FALSE);

//Assert
AssertEquals(Expected := nValueExpected,
             Actual := nValueActual,
             Message := 'nValueActual not returning expected value');
	 
TEST_FINISHED();


TEST('MEMCPY WORD SWAP');
	
//Arrange
nValue := 16#A1B2;
nValueExpected := HOST_TO_BE16(nValue);

//Act
F_MEMCPY(ADR(nValueActual), ADR(nValue), 2, TRUE);

//Assert
AssertEquals(Expected := nValueExpected,
             Actual := nValueActual,
             Message := 'nValueActual not returning expected value');
	 
TEST_FINISHED();
END_METHOD

END_FUNCTION_BLOCK

// ---- Common/Utils/F_Memcpy.TcPOU
(*
	Custom MEMCPY function with a swap flag. 
	If bSwap is true and the length is within the range of 0 to 8, the memcpy operation will be performed with reversed byte order.
*) 
FUNCTION F_Memcpy : UDINT
VAR_INPUT
	destAddr 	: PVOID; //Destination Addr
	srcAddr 	: PVOID; //Source Addr
	n			: UDINT; //Bytes Length
	bSwap		: BOOL; //If TRUE and the length is within the range of 0 to 8, the memcpy operation will be performed with reversed byte order
END_VAR

VAR
	i 			: UDINT;
	aBuffer 	: ARRAY [0..7] OF BYTE;
	nWWORD		: WORD;
	nDWORD		: DWORD;
	nLWORD		: LWORD;
END_VAR

IF NOT bSWAP OR n > 8 THEN
	F_MEMCPY := MEMCPY(destAddr, srcAddr, n);
	RETURN;
END_IF

F_MEMCPY := MEMCPY(ADR(aBuffer), srcAddr, n);

FOR i:= 1 TO n DO	
	MEMCPY(destAddr + i - 1, ADR(aBuffer) + n - i, 1);
END_FOR

END_FUNCTION

// ---- Tests/Components/FB_Heater_Test.TcPOU
FUNCTION_BLOCK FB_Heater_Test EXTENDS TcUnit.FB_TestSuite

TestState();
TestLimits();
TestValueChange();

METHOD TestLimits : REFERENCE TO FB_Test
VAR
	fbHeater : FB_Heater();
END_VAR
TEST('Limit Min FALSE');
fbHeater.fHeatingSpeed := 0;
fbHeater.fCoolingSpeed := 0;
fbHeater.fLimitMin := 20;
fbHeater.fValue := 30;

fbHeater();

AssertFALSE(fbHeater.bIsLimitMin, 'State is not correct');	 
TEST_FINISHED();

TEST('Limit Min TRUE');
fbHeater.fHeatingSpeed := 0;
fbHeater.fCoolingSpeed := 0;
fbHeater.fLimitMin := 20;
fbHeater.fValue := 20;

fbHeater();

AssertTRUE(fbHeater.bIsLimitMin, 'State is not correct');	 
TEST_FINISHED();

TEST('Limit Max FALSE');
fbHeater.fHeatingSpeed := 0;
fbHeater.fCoolingSpeed := 0;
fbHeater.fLimitMax := 60;
fbHeater.fValue := 59.9999;

fbHeater();

AssertFALSE(fbHeater.bIsLimitMax, 'State is not correct');	 
TEST_FINISHED();

TEST('Limit Max TRUE');
fbHeater.fHeatingSpeed := 0;
fbHeater.fCoolingSpeed := 0;
fbHeater.fLimitMax := 60;
fbHeater.fValue := 60;

fbHeater();

AssertTRUE(fbHeater.bIsLimitMax, 'State is not correct');	 
TEST_FINISHED();
END_METHOD

METHOD TestState : REFERENCE TO FB_Test
VAR
	fbHeater : FB_Heater();
END_VAR
TEST('State Enable');
fbHeater.bEnable := TRUE;	
fbHeater();
AssertTRUE(fbHeater.bEnabled, 'State is not correct');	 
TEST_FINISHED();

TEST('State Disable');
fbHeater.bEnable := TRUE;	
fbHeater();
fbHeater.bEnable := FALSE;
fbHeater();	
AssertFALSE(fbHeater.bEnabled, 'State is not correct');	 
TEST_FINISHED();
END_METHOD

METHOD TestValueChange : REFERENCE TO FB_Test
VAR
	fbHeater : FB_Heater();
	fResult : REAL;	
	fExpected : REAL;
	bExpected : BOOL;
	fInitValue : REAL;
	nCycleCount : INT;
END_VAR
TEST('Value Up Disable');

fInitValue := 30;

fbHeater.bEnable := FALSE;
fbHeater.fValue := fInitValue;
fbHeater.fHeatingSpeed := 10;
fbHeater.fCoolingSpeed := 0;

fbHeater();

fResult := fbHeater.fValue;
fExpected := fInitValue;

AssertEquals(Expected := fExpected,
             Actual := fResult,
             Message := 'Result value is not correct');	
	 
TEST_FINISHED();


TEST('Value Up Enable');

fInitValue := 30;

fbHeater.bEnable := TRUE;
fbHeater.fValue := fInitValue;
fbHeater.fHeatingSpeed := 10;
fbHeater.fCoolingSpeed := 0;

fbHeater();

fResult := fbHeater.fValue;
fExpected := fInitValue + 10 * GVL_Core.fbSystem.fDeltaTime;

AssertEquals(Expected := fExpected,
             Actual := fResult,
             Message := 'Result value is not correct');	
	 
TEST_FINISHED();


TEST('Value Down Disable');

fInitValue := 30;

fbHeater.bEnable := FALSE;
fbHeater.fValue := fInitValue;
fbHeater.fHeatingSpeed := 10;
fbHeater.fCoolingSpeed := 0;

fbHeater();

fResult := fbHeater.fValue;
fExpected := fInitValue;

AssertEquals(Expected := fExpected,
             Actual := fResult,
             Message := 'Result value is not correct');	
	 
TEST_FINISHED();


TEST('Value Down Enable');

fInitValue := 30;

fbHeater.bEnable := TRUE;
fbHeater.fValue := fInitValue;
fbHeater.fHeatingSpeed := 20;
fbHeater.fCoolingSpeed := 30;

fbHeater();

fResult := fbHeater.fValue;
fExpected := fInitValue - 10 * GVL_Core.fbSystem.fDeltaTime;

AssertEquals(Expected := fExpected,
             Actual := fResult,
             Message := 'Result value is not correct');	
	 
TEST_FINISHED();

TEST('Value Cooling');

fInitValue := 30;

fbHeater.bEnable := FALSE;
fbHeater.fValue := fInitValue;
fbHeater.fHeatingSpeed := 0;
fbHeater.fCoolingSpeed := 10;

fbHeater();

fResult := fbHeater.fValue;
fExpected := fInitValue - 10 * GVL_Core.fbSystem.fDeltaTime;

AssertEquals(Expected := fExpected,
             Actual := fResult,
             Message := 'Result value is not correct');	
	 
TEST_FINISHED();
END_METHOD

END_FUNCTION_BLOCK

// ---- Common/Components/FB_Heater.TcPOU
FUNCTION_BLOCK FB_Heater
VAR_INPUT
	bEnable 		: BOOL;	
	fHeatingSpeed 	: REAL := 1; //[*/s]
	fCoolingSpeed 	: REAL := 1; //[*/s]
	fLimitMin 		: REAL := 0; //[*]
	fLimitMax 		: REAL := 100; //[*]
END_VAR

VAR_OUTPUT
	bEnabled 		: BOOL;
	bIsLimitMin		: BOOL;
	bIsLimitMax		: BOOL;	
END_VAR

VAR
	_fValue 		: REAL; //[*]
END_VAR

InitRun();

bEnabled := bEnable;

_fValue := _fValue - fCoolingSpeed * GVL_Core.fbSystem.fDeltaTime;

IF bEnable THEN
	_fValue := _fValue + fHeatingSpeed * GVL_Core.fbSystem.fDeltaTime;
END_IF

bIsLimitMin := _fValue <= fLimitMin;
bIsLimitMax := _fValue >= fLimitMax;
_fValue := LIMIT(fLimitMin, _fValue, fLimitMax);

PROPERTY fValue : REAL
GET
fValue := _fValue;
END_GET
SET
_fValue := fValue;
END_SET
END_PROPERTY

METHOD INTERNAL InitRun
VAR_INST
	bInitRun : BOOL := TRUE;
END_VAR
IF NOT bInitRun THEN RETURN; END_IF
bInitRun := FALSE;
END_METHOD

END_FUNCTION_BLOCK

// ---- Tests/Components/FB_MoveVelocity_Test.TcPOU
FUNCTION_BLOCK FB_MoveVelocity_Test EXTENDS TcUnit.FB_TestSuite

TestCaseMove('Set Init',0, 0, 1000, 1000, TRUE);

TestCaseMove('Set Valid Motion_1',0, 1000, 1000, 1000, FALSE);
TestCaseMove('Set Valid Motion_2',0, 100, 1000, 1000, FALSE);
TestCaseMove('Set Valid Motion_3',0, 10, 1000, 1000, TRUE);	
TestCaseMove('Set Valid Motion_4',0, -1000, -1000, -1000, FALSE);
TestCaseMove('Set Valid Motion_5',0, -100, -1000, -1000, FALSE);
TestCaseMove('Set Valid Motion_6',0, -10, -1000, -1000, TRUE);

TestCaseMove('Set 2Zone Motion_1',-5, 1000, 1000, 1000, FALSE);
TestCaseMove('Set 2Zone Motion_2',-5, 100, 1000, 1000, FALSE);
TestCaseMove('Set 2Zone Motion_3',-5, 10, 2000, 2000, TRUE);	
TestCaseMove('Set 2Zone Motion_4',5, -1000, -1000, -1000, FALSE);
TestCaseMove('Set 2Zone Motion_5',5, -100, -1000, -1000, FALSE);
TestCaseMove('Set 2Zone Motion_6',5, -10, -2000, -2000, TRUE);

TestCaseMove('Set Dirty Motion_1',0, 10, 0.001, 0.001, FALSE);
TestCaseMove('Set Dirty Motion_2',0, 10, 0, 0, FALSE);
TestCaseMove('Set Dirty Motion_3',0, 10, 1E+12, 1E+12, TRUE);	
TestCaseMove('Set Dirty Motion_4',0, -1E+3, 1E+12, 1E+12, TRUE);	

TestCaseMove('Set Dirty ACC/DEC_1',0, 1000, -1000, -1000, FALSE);
TestCaseMove('Set Dirty ACC/DEC_2',0, 100, -1000, -1000, FALSE);
TestCaseMove('Set Dirty ACC/DEC_3',0, 10, -1000, -1000, TRUE);
TestCaseMove('Set Dirty ACC/DEC_4',0, -1000, 1000, 1000, FALSE);
TestCaseMove('Set Dirty ACC/DEC_5',0, -100, 1000, 1000, FALSE);
TestCaseMove('Set Dirty ACC/DEC_6',0, -10, 1000, 1000, TRUE);

METHOD TestCaseMove
VAR_INPUT
	sName 				: T_MaxString;
	fInitVelocity 		: REAL;
	fVelocity 			: REAL;
	fAcceleration 		: REAL;
	fDeceleration 		: REAL;
	bExpected 			: BOOL;
END_VAR

VAR
	fbMoveVelocity 		: FB_MoveVelocity;
	nCycleCount 		: INT;
	bResult 			: BOOL;
	fResult 			: REAL;
	fAcc 				: REAL;
	fExpectedAcc 		: REAL := 0;
END_VAR
TEST(sName);
	
fbMoveVelocity.fVelocity := fInitVelocity;

FOR nCycleCount := 0 TO 10 DO
    fbMoveVelocity(fTargetVelocity := fVelocity, fAccMax := fAcceleration, fDecMax := fDeceleration);
END_FOR;

bResult := fbMoveVelocity.bIsReached;
fResult := fbMoveVelocity.fVelocity;
fAcc := fbMoveVelocity.fAcc;

AssertEquals(Expected := bExpected,
             Actual := bResult,
             Message := 'Value is not reached');	
			 
IF bExpected THEN
	AssertEquals(Expected := fVelocity,
             Actual := fResult,
             Message := 'Velocity value is not correct');	
	AssertEquals(Expected := fExpectedAcc,
             Actual := fAcc,
             Message := 'Acc value is not correct');	
END_IF
	 
TEST_FINISHED();
END_METHOD

END_FUNCTION_BLOCK

// ---- Common/Components/FB_MoveVelocity.TcPOU
(* 
	FB_MoveVelocity: Adjusts the drive's velocity based on target velocity, acceleration, and deceleration
*)
FUNCTION_BLOCK FB_MoveVelocity
VAR_INPUT
	fTargetVelocity 	: REAL;
	fAccMax 			: REAL;
	fDecMax 			: REAL;
END_VAR

VAR
	_fVelocity 			: REAL;	
	_fAcc 				: REAL;
	_bIsReached			: BOOL;
	_fVelocityTolerance	: REAL;
END_VAR

_bIsReached := FALSE;
IF _fAcc = 0 THEN
	IF ABS(fAccMax) > ABS(fDecMax) THEN
		_fVelocityTolerance := ABS(fAccMax) * GVL_Core.fbSystem.fDeltaTime * GVL_Core.fbSystem.fTimeScaling;
	ELSE
		_fVelocityTolerance := ABS(fDecMax) * GVL_Core.fbSystem.fDeltaTime * GVL_Core.fbSystem.fTimeScaling;
	END_IF
ELSE
	_fVelocityTolerance := ABS(_fAcc) * GVL_Core.fbSystem.fDeltaTime * GVL_Core.fbSystem.fTimeScaling;
END_IF	

(* Calculate acceleration *)
//Hold velocity (velocity reached)
IF F_Compare(fVelocity, fTargetVelocity, _fVelocityTolerance) THEN
	_fAcc := 0;
	_fVelocity := fTargetVelocity;
	_bIsReached := TRUE;
	RETURN;
END_IF

IF _fVelocity - fTargetVelocity > _fVelocityTolerance THEN
	//Decelerate
	IF _fVelocity < 0 THEN
		_fAcc := -ABS(fAccMax);
	ELSE
		_fAcc := -ABS(fDecMax);
	END_IF
 ELSIF _fVelocity - fTargetVelocity < -_fVelocityTolerance THEN
	//Accelerate
	IF _fVelocity < 0 THEN
		_fAcc := ABS(fDecMax);
	ELSE
		_fAcc := ABS(fAccMax);
	END_IF
END_IF

_fVelocity := _fVelocity + _fAcc * GVL_Core.fbSystem.fDeltaTime * GVL_Core.fbSystem.fTimeScaling;
_bIsReached := F_Compare(_fVelocity, fTargetVelocity, _fVelocityTolerance);

(* 
	bIsReached: TRUE if the current velocity has reached the target velocity 
*)
PROPERTY bIsReached : BOOL
GET
bIsReached := THIS^._bIsReached;
END_GET
END_PROPERTY

(*
    Actual Drive Acceleration
	
	The fAcc property provides the current acceleration for the drive.
*)
PROPERTY fAcc : REAL
GET
fAcc := THIS^._fAcc;
END_GET
SET
THIS^._fAcc := fAcc;
END_SET
END_PROPERTY

(*
    Actual Drive Velocity
	
	The fVelocity property provides the current velocity for the drive.
*)
PROPERTY fVelocity : REAL
GET
fVelocity := THIS^._fVelocity;
END_GET
SET
THIS^._fVelocity := fVelocity;
END_SET
END_PROPERTY

END_FUNCTION_BLOCK

// ---- Tests/Components/FB_MoveAbsolute_Test.TcPOU
FUNCTION_BLOCK FB_MoveAbsolute_Test EXTENDS TcUnit.FB_TestSuite

TestCaseMoveTo('Set Init', fInitPosition := 0, fInitVelocity := 0, fPosition := 0, fVelocity := 100, fAcceleration := 1E+6, fDeceleration := 1E+6, TRUE);

TestCaseMoveTo('Set Valid Motion_1', fInitPosition := 0, fInitVelocity := 0, fPosition := 1, fVelocity := 1000, fAcceleration := 1E+6, fDeceleration := 1E+6, TRUE);
TestCaseMoveTo('Set Valid Motion_2', fInitPosition := 0, fInitVelocity := 0, fPosition := 10, fVelocity := 1000, fAcceleration := 1E+6, fDeceleration := 1E+6, TRUE);
TestCaseMoveTo('Set Valid Motion_3', fInitPosition := 0, fInitVelocity := 0, fPosition := 100, fVelocity := 1000, fAcceleration := 1E+6, fDeceleration := 1E+6, FALSE);
TestCaseMoveTo('Set Valid Motion_4', fInitPosition := 0, fInitVelocity := 0, fPosition := 1000, fVelocity := 1000, fAcceleration := 1E+6, fDeceleration := 1E+6, FALSE);

TestCaseMoveTo('Set 2Zone Motion_1', fInitPosition := -5, fInitVelocity := 0, fPosition := 1, fVelocity := 1000, fAcceleration := 1E+6, fDeceleration := 1E+6, TRUE);
TestCaseMoveTo('Set 2Zone Motion_2', fInitPosition := -5, fInitVelocity := 0, fPosition := 5, fVelocity := 1000, fAcceleration := 1E+6, fDeceleration := 1E+6, TRUE);
TestCaseMoveTo('Set 2Zone Motion_3', fInitPosition := 5, fInitVelocity := 0, fPosition := -1, fVelocity := 1000, fAcceleration := 1E+6, fDeceleration := 1E+6, TRUE);
TestCaseMoveTo('Set 2Zone Motion_4', fInitPosition := 5, fInitVelocity := 0, fPosition := -5, fVelocity := 1000, fAcceleration := 1E+6, fDeceleration := 1E+6, TRUE);

TestCaseMoveTo('Set Dirty Motion_1', fInitPosition := 0, fInitVelocity := 0, fPosition := 1, fVelocity := -1000, fAcceleration := -1E+6, fDeceleration := -1E+6, TRUE);
TestCaseMoveTo('Set Dirty Motion_2', fInitPosition := 0, fInitVelocity := 0, fPosition := 10, fVelocity := -1000, fAcceleration := -1E+6, fDeceleration := -1E+6, TRUE);
TestCaseMoveTo('Set Dirty Motion_3', fInitPosition := 0, fInitVelocity := 0, fPosition := 100, fVelocity := -1000, fAcceleration := -1E+6, fDeceleration := -1E+6, FALSE);
TestCaseMoveTo('Set Dirty Motion_4', fInitPosition := 0, fInitVelocity := 0, fPosition := 1000, fVelocity := -1000, fAcceleration := -1E+6, fDeceleration := -1E+6, FALSE);

TestCaseMoveTo('Set Init Velocity_1', fInitPosition := 0, fInitVelocity := 1000, fPosition := 1, fVelocity := 1000, fAcceleration := 1E+6, fDeceleration := 1E+6, TRUE);
TestCaseMoveTo('Set Init Velocity_2', fInitPosition := 0, fInitVelocity := 1000, fPosition := 10, fVelocity := 1000, fAcceleration := 1E+6, fDeceleration := 1E+6, TRUE);
TestCaseMoveTo('Set Init Velocity_3', fInitPosition := 0, fInitVelocity := 1000, fPosition := 100, fVelocity := 1000, fAcceleration := 1E+6, fDeceleration := 1E+6, FALSE);
TestCaseMoveTo('Set Init Velocity_4', fInitPosition := 0, fInitVelocity := 1000, fPosition := 1000, fVelocity := 1000, fAcceleration := 1E+6, fDeceleration := 1E+6, FALSE);

TestCaseMoveTo('Set Init Position_1', fInitPosition := 1, fInitVelocity := 1000, fPosition := 1, fVelocity := 1000, fAcceleration := 1E+6, fDeceleration := 1E+6, TRUE);
TestCaseMoveTo('Set Init Position_2', fInitPosition := 10, fInitVelocity := 1000, fPosition := 10, fVelocity := 1000, fAcceleration := 1E+6, fDeceleration := 1E+6, TRUE);
TestCaseMoveTo('Set Init Position_3', fInitPosition := 100, fInitVelocity := 1000, fPosition := 100, fVelocity := 1000, fAcceleration := 1E+6, fDeceleration := 1E+6, TRUE);
TestCaseMoveTo('Set Init Position_4', fInitPosition := 1000, fInitVelocity := 1000, fPosition := 1000, fVelocity := 1000, fAcceleration := 1E+6, fDeceleration := 1E+6, TRUE);

METHOD TestCaseMoveTo : REFERENCE TO FB_Test
VAR_INPUT
	sName 				: T_MaxString;
	fInitPosition 		: REAL;
	fInitVelocity 		: REAL;
	fPosition 			: REAL;	
	fVelocity 			: REAL; 
	fAcceleration 		: REAL; 
	fDeceleration 		: REAL;	
	bExpected 			: BOOL;
END_VAR

VAR
	fbMoveAbsolute 		: FB_MoveAbsolute;
	nCycleCount 		: INT;
	bResult 			: BOOL;
	fResult 			: REAL;
	fVel 				: REAL;
	fExpectedVel 		: REAL := 0;
END_VAR
TEST(sName);

fbMoveAbsolute.fPosition := fInitPosition;
fbMoveAbsolute.fVelocity := fInitVelocity;

FOR nCycleCount := 0 TO 10 DO
    fbMoveAbsolute( fTargetPosition:= fPosition, 
					fTargetVelocity := fVelocity, 
					fAccMax := fAcceleration, 
					fDecMax := fDeceleration);
END_FOR

bResult := fbMoveAbsolute.bIsReached;
fResult := fbMoveAbsolute.fPosition;
fVel := fbMoveAbsolute.fVelocity;

AssertEquals(Expected := bExpected,
             Actual := bResult,
             Message := 'Value is not reached');

IF bExpected THEN
	AssertEquals(Expected := fPosition,
             Actual := fResult,
             Message := 'Position value is not correct');	
	AssertEquals(Expected := fExpectedVel,
             Actual := fVel,
             Message := 'Velocity value is not correct');	
END_IF
	 
TEST_FINISHED();
END_METHOD

END_FUNCTION_BLOCK

// ---- Common/Components/FB_MoveAbsolute.TcPOU
(* 
	FB_MoveAbsolute: Controls absolute movement using target position, velocity, acceleration, and deceleration. 
*)
FUNCTION_BLOCK FB_MoveAbsolute 
VAR_INPUT
	fTargetPosition 	: REAL;
	fTargetVelocity 	: REAL; 
	fAccMax 			: REAL; 
	fDecMax 			: REAL;	
	fTolerance			: REAL := 1E-6;	
END_VAR

VAR
	_fVelocity 			: REAL;
	_fPosition 			: REAL;
	_bIsReached			: BOOL;
END_VAR

fTargetVelocity := ABS(fTargetVelocity); 
fAccMax := ABS(fAccMax);
fDecMax := -ABS(fDecMax);

IF F_Compare(fTargetPosition, _fPosition, fTolerance) THEN
	_fVelocity := 0;
	_fPosition := fTargetPosition;
	_bIsReached := TRUE;	
ELSE
	(* Calculate velocity and position *)
	IF fTargetPosition > _fPosition THEN		
		IF _fVelocity < 0 THEN
			_fVelocity := MIN(_fVelocity - fDecMax * GVL_Core.fbSystem.fDeltaTime * GVL_Core.fbSystem.fTimeScaling, fTargetVelocity);
		ELSE
			IF _fVelocity > fTargetVelocity THEN
				_fVelocity := MAX(_fVelocity + fDecMax * GVL_Core.fbSystem.fDeltaTime * GVL_Core.fbSystem.fTimeScaling, fTargetVelocity);
			ELSE
				_fVelocity := MIN(_fVelocity + fAccMax * GVL_Core.fbSystem.fDeltaTime * GVL_Core.fbSystem.fTimeScaling, fTargetVelocity);
			END_IF

			_fVelocity := MIN(SQRT((_fPosition - fTargetPosition) * 2.0 * fDecMax - 1.5 * GVL_Core.fbSystem.fDeltaTime * GVL_Core.fbSystem.fTimeScaling * fDecMax), _fVelocity);
		END_IF

		_fPosition := _fPosition + MIN(_fVelocity * GVL_Core.fbSystem.fDeltaTime * GVL_Core.fbSystem.fTimeScaling, fTargetPosition - _fPosition);	
	ELSE		
		IF _fVelocity > 0 THEN
			_fVelocity := MAX(_fVelocity + fDecMax * GVL_Core.fbSystem.fDeltaTime * GVL_Core.fbSystem.fTimeScaling, -fTargetVelocity);
		ELSE
			IF _fVelocity < -fTargetVelocity THEN
				_fVelocity := MIN(_fVelocity - fDecMax * GVL_Core.fbSystem.fDeltaTime * GVL_Core.fbSystem.fTimeScaling, -fTargetVelocity);
			ELSE				
				_fVelocity := MAX(_fVelocity - fAccMax * GVL_Core.fbSystem.fDeltaTime * GVL_Core.fbSystem.fTimeScaling, -fTargetVelocity);
			END_IF
			
			_fVelocity := MAX(-SQRT((_fPosition - fTargetPosition) * 2.0 * -fDecMax - 1.5 * GVL_Core.fbSystem.fDeltaTime * GVL_Core.fbSystem.fTimeScaling * fDecMax), _fVelocity);
	   END_IF

		_fPosition := _fPosition + MAX(_fVelocity * GVL_Core.fbSystem.fDeltaTime * GVL_Core.fbSystem.fTimeScaling, fTargetPosition - _fPosition);	
	END_IF;
	
	_bIsReached := FALSE;		
END_IF;

(*
    Indicates whether the drive has reached its target position.

    This property reflects the internal state of the drive control system.
    It returns TRUE if the drive has achieved the desired position within the specified
    tolerance limits; otherwise, it returns FALSE.
*)
PROPERTY bIsReached : BOOL
GET
bIsReached := THIS^._bIsReached;
END_GET
END_PROPERTY

(*
    Actual Drive Position
	
	The fPosition property provides the current position for the drive.
*)
PROPERTY fPosition : REAL
GET
fPosition := _fPosition;
END_GET
SET
_fPosition := fPosition;
END_SET
END_PROPERTY

(*
    Actual Drive Velocity
	
	The fVelocity property provides the current velocity for the drive.
*)
PROPERTY fVelocity : REAL
GET
fVelocity := _fVelocity;
END_GET
SET
_fVelocity := fVelocity;
END_SET
END_PROPERTY

END_FUNCTION_BLOCK

// ---- Tests/Components/FB_DriveControl_Test.TcPOU
FUNCTION_BLOCK FB_DriveControl_Test EXTENDS TcUnit.FB_TestSuite

TestCaseMoveVelocityLimits();
TestProperties();

TestCaseMoveVelocity('Velocity Zero', 0, 0, TRUE);

TestCaseMoveVelocity('Target Positiv Velocity_1', 0, 10, TRUE);
TestCaseMoveVelocity('Target Positiv Velocity_2', 90, 100, TRUE);
TestCaseMoveVelocity('Target Positiv Velocity_3', 990, 1000, TRUE);
TestCaseMoveVelocity('Target Positiv Velocity_4', 50, 100, FALSE);
TestCaseMoveVelocity('Target Positiv Velocity_5', 500, 1000, FALSE);

TestCaseMoveVelocity('Target Negative Velocity_1', 0, -10, TRUE);
TestCaseMoveVelocity('Target Negative Velocity_2', -90, -100, TRUE);
TestCaseMoveVelocity('Target Negative Velocity_3', -990, -1000, TRUE);
TestCaseMoveVelocity('Target Negative Velocity_4', -50, -100, FALSE);
TestCaseMoveVelocity('Target Negative Velocity_5', -500, -1000, FALSE);

TestCaseMoveAbsolute('Move Positive Absolute_1', 0, 1, 1000, TRUE);
TestCaseMoveAbsolute('Move Positive Absolute_2', 0, 10, 1000, TRUE);
TestCaseMoveAbsolute('Move Positive Absolute_3', 0, 100, 1000, FALSE);
TestCaseMoveAbsolute('Move Positive Absolute_4', 0, 1000, 1000, FALSE);

TestCaseMoveAbsolute('Move Positive Absolute_11', 50, 51, 1000, TRUE);
TestCaseMoveAbsolute('Move Positive Absolute_12', 50, 60, 1000, TRUE);
TestCaseMoveAbsolute('Move Positive Absolute_13', -50, -49, 1000, TRUE);
TestCaseMoveAbsolute('Move Positive Absolute_14', -50, -40, 1000, TRUE);

TestCaseMoveAbsolute('Move Negative Absolute_1', 0, -1, 1000, TRUE);
TestCaseMoveAbsolute('Move Negative Absolute_2', 0, -10, 1000, TRUE);
TestCaseMoveAbsolute('Move Negative Absolute_3', 0, -100, 1000, FALSE);
TestCaseMoveAbsolute('Move Negative Absolute_4', 0, -1000, 1000, FALSE);

TestCaseMoveAbsolute('Move Negative Absolute_11', -50, -51, 1000, TRUE);
TestCaseMoveAbsolute('Move Negative Absolute_12', -50, -60, 1000, TRUE);
TestCaseMoveAbsolute('Move Negative Absolute_13', 50, 49, 1000, TRUE);
TestCaseMoveAbsolute('Move Negative Absolute_14', 50, 40, 1000, TRUE);

TestStop();

METHOD TestCaseMoveAbsolute
VAR_INPUT
	sName 				: T_MaxString;
	fInitPosition 		: REAL;
	fTargetPosition 	: REAL;
	fTargetVelocity 	: REAL;
	bExpected 			: BOOL;
END_VAR

VAR
	fbDriveControl 		: FB_DriveControl;
	nCycleCount 		: INT;
	bResult 			: BOOL;
	fResult 			: REAL;
	fVel 				: REAL;
	fExpectedVel 		: REAL := 0;
END_VAR
TEST(sName);

fbDriveControl.fPosition := fInitPosition;

FOR nCycleCount := 0 TO 10 DO
    fbDriveControl.MoveAbsolute(fTargetPosition, fTargetVelocity, 1E+6, 1E+6);
END_FOR

bResult := fbDriveControl.bIsPositionReached;
fResult := fbDriveControl.fPosition;
fVel := fbDriveControl.fVelocity;

AssertEquals(Expected := bExpected,
             Actual := bResult,
             Message := 'Position is not reached');

IF bExpected THEN
	AssertEquals(Expected := fTargetPosition,
             Actual := fResult,
             Message := 'Position value is not correct');	
	AssertEquals(Expected := fExpectedVel,
             Actual := fVel,
             Message := 'Velocity value is not correct');	
END_IF
	 
TEST_FINISHED();
END_METHOD

METHOD TestCaseMoveVelocity
VAR_INPUT
	sName 				: T_MaxString;
	fInitVelocity 		: REAL;
	fTargetVelocity 	: REAL;
	bExpected 			: BOOL;
END_VAR

VAR
	fbDriveControl 		: FB_DriveControl;
	nCycleCount 		: INT;
	bResult 			: BOOL;	
	fResult 			: REAL;	
END_VAR
TEST(sName);

fbDriveControl.fVelocity := fInitVelocity;

FOR nCycleCount := 0 TO 10 DO
    fbDriveControl.MoveVelocity(fTargetVelocity, 1000, 1000);
END_FOR;

fResult := fbDriveControl.fVelocity;

IF bExpected THEN
	AssertEquals(Expected := fTargetVelocity,
             Actual := fResult,
             Message := 'Velocity value is not correct');
ELSE
	bResult := F_Compare(fbDriveControl.fVelocity, fTargetVelocity, 1E-6);
	AssertFALSE(bResult, 'Not Expected Velocity');	 	
END_IF

TEST_FINISHED();
END_METHOD

METHOD TestCaseMoveVelocityLimits
VAR
	fbDriveControl 		: FB_DriveControl;
	nCycleCount 		: INT;
	bResult 			: BOOL;	
	fResult 			: REAL;	
	fExpected 			: REAL;
END_VAR
TEST('Position Limit Min');

fExpected := 0;
fbDriveControl.fPositionLimitMin := -10;
fbDriveControl.fPosition := -10;

fbDriveControl.MoveVelocity(1000, 1000, 1000);
fResult := fbDriveControl.fVelocity;

AssertEquals(Expected := fExpected,
             Actual := fResult,
             Message := 'Velocity value is not limited');

TEST_FINISHED();

TEST('Position Limit Max');

fExpected := 0;
fbDriveControl.fPositionLimitMax := 10;
fbDriveControl.fPosition := 10;

fbDriveControl.MoveVelocity(1000, 1000, 1000);
fResult := fbDriveControl.fVelocity;

AssertEquals(Expected := fExpected,
             Actual := fResult,
             Message := 'Velocity value is not limited');

TEST_FINISHED();
END_METHOD

METHOD TestProperties
VAR
	fbDriveControl 		: FB_DriveControl;
	fResult 			: REAL;
	fExpected 			: REAL;
END_VAR
TEST('Test Property: fAccMax');
fExpected := 10;
fbDriveControl.fAccMax := fExpected;
fResult := fbDriveControl.fAccMax;

AssertEquals(Expected := fExpected,
             Actual := fResult,
             Message := 'Property value is not correct');
TEST_FINISHED();

TEST('Test Property: fPositionLimitMin');
fExpected := 10;
fbDriveControl.fPositionLimitMin := fExpected;
fResult := fbDriveControl.fPositionLimitMin;

AssertEquals(Expected := fExpected,
             Actual := fResult,
             Message := 'Property value is not correct');
TEST_FINISHED();

TEST('Test Property: fPositionLimitMax');
fExpected := 10;
fbDriveControl.fPositionLimitMax := fExpected;
fResult := fbDriveControl.fPositionLimitMax;

AssertEquals(Expected := fExpected,
             Actual := fResult,
             Message := 'Property value is not correct');
TEST_FINISHED();

TEST('Test Property: fTolerance');
fExpected := 10;
fbDriveControl.fTolerance := fExpected;
fResult := fbDriveControl.fTolerance;

AssertEquals(Expected := fExpected,
             Actual := fResult,
             Message := 'Property value is not correct');
TEST_FINISHED();

TEST('Test Property: fPosition');
fExpected := 10;
fbDriveControl.fPosition := fExpected;
fResult := fbDriveControl.fPosition;

AssertEquals(Expected := fExpected,
             Actual := fResult,
             Message := 'Property value is not correct');
TEST_FINISHED();
END_METHOD

METHOD TestStop : REFERENCE TO FB_Test
VAR
	fbDriveControl 		: FB_DriveControl;
	nCycleCount 		: INT;
	bResult 			: BOOL;
	fResult 			: REAL;
	fExpected 			: REAL;
END_VAR
TEST('Stop');

fbDriveControl.fVelocity := -10; 

bResult := fbDriveControl.bIsMoving;
AssertTrue(bResult, 'Expected Drive in motion');

FOR nCycleCount := 0 TO 10 DO
    fbDriveControl.Stop(1E6);
END_FOR

bResult := fbDriveControl.bIsMoving;
AssertFalse(bResult, 'Expected Drive is stopped');

fExpected := 0;
fResult := fbDriveControl.fVelocity;
AssertEquals(Expected := fExpected,
             Actual := fResult,
             Message := 'fVelocity value is not correct');

TEST_FINISHED();
END_METHOD

END_FUNCTION_BLOCK

// ---- Common/Components/FB_DriveControl.TcPOU
(*
	FB_DriveControl manages drive operations by integrating absolute position and velocity control.
    It encapsulates the functionalities of FB_MoveAbsolute for absolute movement and FB_MoveVelocity
    for velocity-based control.
*)
FUNCTION_BLOCK FB_DriveControl
VAR
	_fbMoveAbsolute 		: FB_MoveAbsolute();
	_fbMoveVelocity			: FB_MoveVelocity();

	_fPosition 				: REAL;
	_fVelocity 				: REAL;		
	_bIsPositionReached 	: BOOL := TRUE;		
	
	_fPositionLimitMin 		: REAL := -1E+12;
	_fPositionLimitMax 		: REAL := 1E+12;
	_fAccMax				: REAL := 1E+12;	
	_fTolerance				: REAL := 1E-6;	
END_VAR

(*
    Indicates whether the drive is currently in motion.

    The bIsMoving property returns TRUE if the drive is actively moving toward its target.
*)
PROPERTY bIsMoving : BOOL
GET
bIsMoving := NOT F_Compare(_fVelocity, 0, 1E-3);
END_GET
END_PROPERTY

(*
    Indicates whether the drive has reached its target position.

    This property reflects the internal state of the drive control system.
    It returns TRUE if the drive has achieved the desired position within the specified
    tolerance limits; otherwise, it returns FALSE.
*)
PROPERTY bIsPositionReached : BOOL
GET
bIsPositionReached := _bIsPositionReached;
END_GET
END_PROPERTY

(*
    Maximum Acceleration Limit

    The fAccMax property represents the maximum acceleration permitted for drive movements.
*)
PROPERTY fAccMax : REAL
GET
fAccMax := _fAccMax;
END_GET
SET
_fAccMax := fAccMax;
END_SET
END_PROPERTY

(*
    Actual Drive Position
	
	The fPosition property provides the current position for the drive.
*)
PROPERTY fPosition : REAL
GET
fPosition := _fPosition;
END_GET
SET
_fPosition := fPosition;
END_SET
END_PROPERTY

(*
    Maximum Position Limit
	
	The fPositionLimitMax property defines the upper boundary for the drive's position.
*)
PROPERTY fPositionLimitMax : REAL
GET
fPositionLimitMax := _fPositionLimitMax;
END_GET
SET
_fPositionLimitMax := fPositionLimitMax;
END_SET
END_PROPERTY

(*
    Minimum  Position Limit
	
	The fPositionLimitMax property defines the lower boundary for the drive's position.
*)
PROPERTY fPositionLimitMin : REAL
GET
fPositionLimitMin := _fPositionLimitMin;
END_GET
SET
_fPositionLimitMin := fPositionLimitMin;
END_SET
END_PROPERTY

(*
    Position Tolerance
	
	The fTolerance property defines the acceptable error range for the drive's position.
*)
PROPERTY fTolerance : REAL
GET
fTolerance := _fTolerance;
END_GET
SET
_fTolerance := fTolerance;
END_SET
END_PROPERTY

(*
    Actual Drive Velocity
	
	The fVelocity property provides the current velocity for the drive.
*)
PROPERTY fVelocity : REAL
GET
fVelocity := _fVelocity;
END_GET
SET
_fVelocity := fVelocity;
END_SET
END_PROPERTY

(* 
    Moves the drive to an absolute position.
    
    The MoveAbsolute method commands the drive to move to a specified absolute position with a given velocity,
    acceleration, and deceleration.
*)
METHOD MoveAbsolute
VAR_INPUT
	fPosition 			: REAL;
	fVelocity			: REAL;
	fAcceleration		: REAL;
	fDeceleration   	: REAL;
END_VAR
_fbMoveAbsolute.fPosition := _fPosition;
_fbMoveAbsolute.fVelocity := _fVelocity;

_fbMoveAbsolute(
	fTargetPosition := LIMIT(_fPositionLimitMin, fPosition, _fPositionLimitMax),
	fTargetVelocity := fVelocity,
	fAccMax := fAcceleration,
	fDecMax := fDeceleration,
	fTolerance := _fTolerance);					

_fVelocity := _fbMoveAbsolute.fVelocity;
_fPosition := _fbMoveAbsolute.fPosition;

_bIsPositionReached := F_Compare(fPosition, _fPosition, _fTolerance);
END_METHOD

(* 
    Moves the drive using velocity control.
    
    The MoveVelocity method commands the drive to move with a specified velocity and controls the acceleration
    and deceleration parameters. It also enforces position limits to prevent the drive from exceeding its boundaries.
*)
METHOD MoveVelocity
VAR_INPUT
	fVelocity 			: REAL;
	fAcceleration 		: REAL;
	fDeceleration 		: REAL;
END_VAR
_fbMoveVelocity.fVelocity := _fVelocity;
_fbMoveVelocity.fTargetVelocity := fVelocity;
_fbMoveVelocity.fAccMax := fAcceleration;
_fbMoveVelocity.fDecMax := fDeceleration;	
	
IF _fPositionLimitMax <> 0 AND _fPositionLimitMin <> 0 THEN
	IF _fPosition >= _fPositionLimitMax OR _fPosition <= _fPositionLimitMin THEN
		_fbMoveVelocity.fTargetVelocity := 0;
		_fbMoveVelocity.fAccMax := _fAccMax;
		_fbMoveVelocity.fDecMax := _fAccMax;
	END_IF		
END_IF
	
_fbMoveVelocity();
	
_fVelocity := _fbMoveVelocity.fVelocity;	

_fPosition := _fPosition + _fVelocity * GVL_Core.fbSystem.fDeltaTime * GVL_Core.fbSystem.fTimeScaling;
_bIsPositionReached := F_Compare(fPosition, _fPosition, _fTolerance);
END_METHOD

(* 
    Stops the drive movement.
    
    The Stop method decelerates the drive until it comes to a complete halt using the specified deceleration.
*)
METHOD Stop
VAR_INPUT
	fDeceleration 	: REAL; 
END_VAR

VAR
	fSign 			: REAL;
	fAbsVelocity 	: REAL;
END_VAR
fSign := F_Sign(_fVelocity);
fAbsVelocity := ABS(_fVelocity);

IF fAbsVelocity > fTolerance THEN
	fAbsVelocity := fAbsVelocity - ABS(fDeceleration) * GVL_Core.fbSystem.fDeltaTime * GVL_Core.fbSystem.fTimeScaling;
	fAbsVelocity := LIMIT(0, fAbsVelocity, 3.402823E+38);
	_fVelocity := fAbsVelocity * fSign;	
ELSE
	_fVelocity := 0;
END_IF
END_METHOD

END_FUNCTION_BLOCK

// ---- Tests/Devices/FB_Button_Test.TcPOU
FUNCTION_BLOCK FB_Button_Test EXTENDS TcUnit.FB_TestSuite
VAR
	_fbButton 		: FB_Button;
	_nExpected 		: BYTE;
	_nResult 		: BYTE;
	_bExpected 		: BOOL;
	_bResult 		: BOOL;
END_VAR

TEST('Set bEnable TRUE');			 
_fbButton.bEnable := TRUE; 
_fbButton();
_nExpected := 1;
_nResult := _fbButton.GetControl();
AssertEquals(Expected := _nExpected,
             Actual := _nResult,
             Message := 'Control value is not correct');	 
TEST_FINISHED();

TEST('Set bEnable FALSE');			 
_fbButton.bEnable := FALSE; 
_fbButton();
_nExpected := 0;
_nResult := _fbButton.GetControl();
AssertEquals(Expected := _nExpected,
             Actual := _nResult,
             Message := 'Control value is not correct');	 
TEST_FINISHED();


TEST('Get bValue FALSE');
_fbButton.SetStatus(0);
_fbButton();
_bExpected := FALSE;
_bResult := _fbButton.bValue;

AssertEquals(Expected := _bExpected,
             Actual := _bResult,
             Message := 'Value is not correct');	
TEST_FINISHED();

TEST('Get bValue TRUE');	
_fbButton.SetStatus(1);
_fbButton();
_bExpected := 1;
_bResult := _fbButton.bValue;
AssertEquals(Expected := _bExpected,
             Actual := _bResult,
             Message := 'Control value is not correct');	 
TEST_FINISHED();

END_FUNCTION_BLOCK

// ---- Devices/Basic/FB_Button.TcPOU
(*
	Default button device.
*)
FUNCTION_BLOCK FB_Button EXTENDS FB_LinkDevice 
VAR_INPUT
	bEnable		: BOOL; //0-Lamp OFF, 1-Lamp ON
END_VAR

VAR_OUTPUT
	bValue		: BOOL; //0-Released, 1-Pressed
END_VAR

SUPER^();
Control.0 := bEnable;
bValue := Status.0;

END_FUNCTION_BLOCK

// ---- Common/Links/FB_LinkDevice.TcPOU
(*
	Base link component with default interface:
	Control BYTE: From TwinCAT >>> To Unity
	Status BYTE: FROM Unity >>> TO TwinCAT		
*)
FUNCTION_BLOCK FB_LinkDevice EXTENDS FB_Base
VAR		
	{attribute 'simulation_interface'}
	Control		AT %Q* : BYTE;
	{attribute 'simulation_interface'}
	Status		AT %I* : BYTE;
END_VAR

SUPER^();

METHOD INTERNAL GetControl : BYTE
GetControl := Control;
END_METHOD

METHOD INTERNAL SetStatus : BOOL
VAR_INPUT
	nStatus : BYTE;
END_VAR
Status := nStatus;
END_METHOD

END_FUNCTION_BLOCK

// ---- Common/System/FB_Base.TcPOU
FUNCTION_BLOCK FB_Base

F_IsSystemValid();

END_FUNCTION_BLOCK

// ---- Common/System/F_IsSystemValid.TcPOU
FUNCTION INTERNAL F_IsSystemValid : BOOL
VAR_STAT
	{attribute 'hide'}
	fbTcConfig		: TC_Config;	
	{attribute 'hide'}
	bIsRequested 	: BOOL;
	{attribute 'hide'}
	bIsSystemValid	: BOOL;
END_VAR

IF NOT bIsRequested THEN
	IF NOT __ISVALIDREF(GVL_Core.refSystem) THEN	
		ADSLOGSTR(msgCtrlMask := ADSLOG_MSGTYPE_ERROR OR ADSLOG_MSGTYPE_MSGBOX, 'OC: %s', 'FB_System can not be found! TwinCAT is switched to Config Mode');
		fbTcConfig(NETID := '', SET := TRUE);
		bIsSystemValid := FALSE;
	ELSE
		bIsSystemValid := TRUE;
	END_IF
END_IF

bIsRequested := TRUE;
F_IsSystemValid := bIsSystemValid;

END_FUNCTION

// ---- Tests/Devices/FB_Switch_Test.TcPOU
FUNCTION_BLOCK FB_Switch_Test EXTENDS TcUnit.FB_TestSuite
VAR
	_fbDevice 		: FB_Switch;
	_nExpected 		: BYTE;
	_nResult 		: BYTE;
END_VAR

TEST('Set nControl');
_nExpected := 255;
_fbDevice.nControl := _nExpected;
_fbDevice();
_nResult := _fbDevice.GetControl();

AssertEquals(Expected := _nExpected,
             Actual := _nResult,
             Message := 'Value is not correct');	
TEST_FINISHED();

TEST('Get nStatus');
_nExpected := 255;
_fbDevice.SetStatus(_nExpected);
_fbDevice();
_nResult := _fbDevice.nStatus;

AssertEquals(Expected := _nExpected,
             Actual := _nResult,
             Message := 'Value is not correct');	
TEST_FINISHED();

END_FUNCTION_BLOCK

// ---- Devices/Basic/FB_Switch.TcPOU
(*
	Default switch device. 	
*)
FUNCTION_BLOCK FB_Switch EXTENDS FB_LinkDevice
VAR_INPUT		
	nControl  			: BYTE;
END_VAR

VAR_OUTPUT
	nStatus  			: BYTE;
END_VAR

SUPER^();
Control := nControl;
nStatus := Status;

END_FUNCTION_BLOCK

// ---- Tests/Devices/FB_Lock_Test.TcPOU
FUNCTION_BLOCK FB_Lock_Test EXTENDS TcUnit.FB_TestSuite
VAR
	_fbLock 		: FB_Lock;
	_nExpected 		: BYTE;
	_nResult 		: BYTE;
	_bExpected 		: BOOL;
	_bResult 		: BOOL;
END_VAR

TEST('Set bEnable TRUE');			 
_fbLock.bLock := TRUE; 
_fbLock();
_nExpected := 1;
_nResult := _fbLock.GetControl();
AssertEquals(Expected := _nExpected,
             Actual := _nResult,
             Message := 'Control value is not correct');	 
TEST_FINISHED();

TEST('Set bEnable FALSE');			 
_fbLock.bLock := FALSE; 
_fbLock();
_nExpected := 0;
_nResult := _fbLock.GetControl();
AssertEquals(Expected := _nExpected,
             Actual := _nResult,
             Message := 'Value is not correct');	 
TEST_FINISHED();


TEST('Get bClosed FALSE');
_fbLock.SetStatus(0);
_fbLock();
_bExpected := FALSE;
_bResult := _fbLock.bClosed;

AssertEquals(Expected := _bExpected,
             Actual := _bResult,
             Message := 'Value is not correct');	
TEST_FINISHED();

TEST('Get bClosed TRUE');	
_fbLock.SetStatus(1);
_fbLock();
_bExpected := 1;
_bResult := _fbLock.bClosed;
AssertEquals(Expected := _bExpected,
             Actual := _bResult,
             Message := 'Value is not correct');	 
TEST_FINISHED();

TEST('Get bLocked FALSE');
_fbLock.SetStatus(0);
_fbLock();
_bExpected := FALSE;
_bResult := _fbLock.bLocked;

AssertEquals(Expected := _bExpected,
             Actual := _bResult,
             Message := 'Value is not correct');	
TEST_FINISHED();

TEST('Get bLocked TRUE');	
_fbLock.SetStatus(2);
_fbLock();
_bExpected := 1;
_bResult := _fbLock.bLocked;
AssertEquals(Expected := _bExpected,
             Actual := _bResult,
             Message := 'Value is not correct');	 
TEST_FINISHED();

TEST('Set nDataIn');
_nExpected := 255;
_fbLock.nControlData := _nExpected;
_fbLock();
_nResult := _fbLock.GetLinkControlData();

AssertEquals(Expected := _nExpected,
             Actual := _nResult,
             Message := 'Value is not correct');	
TEST_FINISHED();

TEST('Get nDataOut');
_nExpected := 255;
_fbLock.SetLinkStatusData(_nExpected);
_fbLock();
_nResult := _fbLock.nStatusData;

AssertEquals(Expected := _nExpected,
             Actual := _nResult,
             Message := 'Value is not correct');	
TEST_FINISHED();

END_FUNCTION_BLOCK

// ---- Devices/Basic/FB_Lock.TcPOU
(*
	Default Lock device
*)
FUNCTION_BLOCK FB_Lock EXTENDS FB_LinkDataByte 
VAR_INPUT
	bLock			: BOOL;
	nControlData	: BYTE;
END_VAR

VAR_OUTPUT	
	bClosed 		: BOOL;
	bLocked 		: BOOL; 
	nStatusData		: BYTE;
END_VAR

SUPER^();
Control.0 := bLock;
ControlData := nControlData;

bClosed := Status.0;
bLocked := Status.1;
nStatusData := StatusData;

END_FUNCTION_BLOCK

// ---- Common/Links/FB_LinkDataByte.TcPOU
(*
	Link component with additional interface:
	Control BYTE: From TwinCAT >>> To Unity	(Default)
	Status BYTE: FROM Unity >>> TO TwinCAT	(Default)	
	ControlData BYTE: From TwinCAT >>> To Unity		
	StatusData BYTE: FROM Unity >>> TO TwinCAT	
*)
FUNCTION_BLOCK FB_LinkDataByte EXTENDS FB_LinkDevice
VAR	
	{attribute 'simulation_interface'}
	ControlData		AT %Q* : BYTE;
	{attribute 'simulation_interface'}
	StatusData		AT %I* : BYTE;
END_VAR

SUPER^();

METHOD INTERNAL GetLinkControlData : BYTE
GetLinkControlData := ControlData;
END_METHOD

METHOD INTERNAL SetLinkStatusData : BOOL
VAR_INPUT
	nStatusData : BYTE;
END_VAR
StatusData := nStatusData;
END_METHOD

END_FUNCTION_BLOCK

// ---- Tests/Devices/FB_Panel_Test.TcPOU
FUNCTION_BLOCK FB_Panel_Test EXTENDS TcUnit.FB_TestSuite
VAR
	_fbPanel 		: FB_Panel;
	_nExpected 		: DWORD;
	_nResult 		: DWORD;
	_bExpected 		: BOOL;
	_bResult 		: BOOL;
END_VAR

TEST('Set nDataIn');
_nExpected := 255;
_fbPanel.nControlData := _nExpected;
_fbPanel();
_nResult := _fbPanel.GetLinkControlData();

AssertEquals(Expected := _nExpected,
             Actual := _nResult,
             Message := 'Value is not correct');	
TEST_FINISHED();

TEST('Get nDataOut');
_nExpected := 255;
_fbPanel.SetLinkStatusData(_nExpected);
_fbPanel();
_nResult := _fbPanel.nStatusData;

AssertEquals(Expected := _nExpected,
             Actual := _nResult,
             Message := 'Value is not correct');	
TEST_FINISHED();

END_FUNCTION_BLOCK

// ---- Devices/Basic/FB_Panel.TcPOU
(*
	Basic panel with extended interface:
	nControl BYTE: From TwinCAT >>> To Unity
	nStatus BYTE: FROM Unity >>> TO TwinCAT	
	nControlData DWORD: From TwinCAT >>> To Unity
	nStatusData DWORD: FROM Unity >>> TO TwinCAT	
*)
FUNCTION_BLOCK FB_Panel EXTENDS FB_LinkDataDWord
VAR_INPUT
	nControlData  			: DWORD;
END_VAR

VAR_OUTPUT	
	nStatusData  			: DWORD;
END_VAR

SUPER^();
ControlData := nControlData;
nStatusData := StatusData;

END_FUNCTION_BLOCK

// ---- Common/Links/FB_LinkDataDWord.TcPOU
(*
	Link component with additional interface:
	Control BYTE: From TwinCAT >>> To Unity	(Default)
	Status BYTE: FROM Unity >>> TO TwinCAT	(Default)
	ControlData DWORD: From TwinCAT >>> To Unity		
	StatusData DWORD: FROM Unity >>> TO TwinCAT		
*)
FUNCTION_BLOCK FB_LinkDataDWord EXTENDS FB_LinkDevice
VAR		
	{attribute 'simulation_interface'}
	ControlData		AT %Q* : DWORD;
	{attribute 'simulation_interface'}
	StatusData		AT %I* : DWORD;
END_VAR

SUPER^();

METHOD INTERNAL GetLinkControlData : DWORD
GetLinkControlData := ControlData;
END_METHOD

METHOD INTERNAL SetLinkStatusData : BOOL
VAR_INPUT
	nStatusData : DWORD;
END_VAR
StatusData := nStatusData;
END_METHOD

END_FUNCTION_BLOCK

// ---- Tests/Devices/FB_Cylinder_Test.TcPOU
FUNCTION_BLOCK FB_Cylinder_Test EXTENDS TcUnit.FB_TestSuite
VAR
	_fbCylinder 	: FB_Cylinder;
	_nExpected 		: BYTE;
	_nResult 		: BYTE;
	_bExpected 		: BOOL;
	_bResult 		: BOOL;
END_VAR

TEST('bRetract FALSE');
_fbCylinder.bRetract := FALSE;
_fbCylinder();
_bExpected := FALSE;
_nResult := _fbCylinder.GetControl();
_bResult := _nResult.0;

AssertEquals(Expected := _bExpected,
             Actual := _bResult,
             Message := 'Control value is not correct');	
TEST_FINISHED();

TEST('bRetract TRUE');
_fbCylinder.bRetract := TRUE;
_fbCylinder();
_bExpected := TRUE;
_nResult := _fbCylinder.GetControl();
_bResult := _nResult.0;

AssertEquals(Expected := _bExpected,
             Actual := _bResult,
             Message := 'Control value is not correct');	
TEST_FINISHED();

TEST('bExtend FALSE');
_fbCylinder.bExtend := FALSE;
_fbCylinder();
_bExpected := FALSE;
_nResult := _fbCylinder.GetControl();
_bResult := _nResult.1;

AssertEquals(Expected := _bExpected,
             Actual := _bResult,
             Message := 'Control value is not correct');	
TEST_FINISHED();

TEST('bExtend TRUE');
_fbCylinder.bExtend := TRUE;
_fbCylinder();
_bExpected := TRUE;
_nResult := _fbCylinder.GetControl();
_bResult := _nResult.1;

AssertEquals(Expected := _bExpected,
             Actual := _bResult,
             Message := 'Control value is not correct');	
TEST_FINISHED();

TEST('bRetracted FALSE');
_fbCylinder.SetStatus(0);
_fbCylinder();
_bExpected := FALSE;
_bResult := _fbCylinder.bRetracted;

AssertEquals(Expected := _bExpected,
             Actual := _bResult,
             Message := 'Control value is not correct');	
TEST_FINISHED();

TEST('bRetracted TRUE');
_fbCylinder.SetStatus(1);
_fbCylinder();
_bExpected := TRUE;
_bResult := _fbCylinder.bRetracted;

AssertEquals(Expected := _bExpected,
             Actual := _bResult,
             Message := 'Control value is not correct');	
TEST_FINISHED();

TEST('bExtended FALSE');
_fbCylinder.SetStatus(0);
_fbCylinder();
_bExpected := FALSE;
_bResult := _fbCylinder.bExtended;

AssertEquals(Expected := _bExpected,
             Actual := _bResult,
             Message := 'Control value is not correct');	
TEST_FINISHED();

TEST('bExtended TRUE');
_fbCylinder.SetStatus(2);
_fbCylinder();
_bExpected := TRUE;
_bResult := _fbCylinder.bExtended;

AssertEquals(Expected := _bExpected,
             Actual := _bResult,
             Message := 'Control value is not correct');	
TEST_FINISHED();

END_FUNCTION_BLOCK

// ---- Devices/Basic/FB_Cylinder.TcPOU
(*
	Default cylinder (valve) device.
*)
FUNCTION_BLOCK FB_Cylinder EXTENDS FB_LinkDevice 
VAR_INPUT
	bRetract : BOOL; //Move to MIN
	bExtend : BOOL; //Move to MAX
END_VAR

VAR_OUTPUT
	bRetracted : BOOL; //Is in MIN
	bExtended : BOOL; //Is in MAX
END_VAR

SUPER^();
bRetracted := Status.0;
bExtended := Status.1;
Control.0 := bRetract;
Control.1 := bExtend;

END_FUNCTION_BLOCK

// ---- Tests/Devices/FB_Device_Test.TcPOU
FUNCTION_BLOCK FB_Device_Test EXTENDS TcUnit.FB_TestSuite
VAR
	_fbDevice 		: FB_Device;
	_nExpected 		: BYTE;
	_nResult 		: BYTE;
END_VAR

TEST('Set nControl');
_nExpected := 255;
_fbDevice.nControl := _nExpected;
_fbDevice();
_nResult := _fbDevice.GetControl();

AssertEquals(Expected := _nExpected,
             Actual := _nResult,
             Message := 'Value is not correct');	
TEST_FINISHED();

TEST('Get nStatus');
_nExpected := 255;
_fbDevice.SetStatus(_nExpected);
_fbDevice();
_nResult := _fbDevice.nStatus;

AssertEquals(Expected := _nExpected,
             Actual := _nResult,
             Message := 'Value is not correct');	
TEST_FINISHED();

END_FUNCTION_BLOCK

// ---- Devices/Basic/FB_Device.TcPOU
(*
	Basic device with default interface:
	nControl BYTE: From TwinCAT >>> To Unity
	nStatus BYTE: FROM Unity >>> TO TwinCAT		
*)
FUNCTION_BLOCK FB_Device EXTENDS FB_LinkDevice
VAR_INPUT		
	nControl  			: BYTE;
END_VAR

VAR_OUTPUT
	nStatus  			: BYTE;
END_VAR

SUPER^();
Control := nControl;
nStatus := Status;

END_FUNCTION_BLOCK

// ---- Tests/Devices/FB_DeviceByte_Test.TcPOU
FUNCTION_BLOCK FB_DeviceByte_Test EXTENDS TcUnit.FB_TestSuite
VAR
	_fbDevice : FB_DeviceByte;
	_nExpected : BYTE;
	_nResult : BYTE;
END_VAR

TEST('Set nControl');
_nExpected := 255;
_fbDevice.nControl := _nExpected;
_fbDevice();
_nResult := _fbDevice.GetControl();

AssertEquals(Expected := _nExpected,
             Actual := _nResult,
             Message := 'Value is not correct');	
TEST_FINISHED();

TEST('Set nDataIn');
_nExpected := 255;
_fbDevice.nControlData := _nExpected;
_fbDevice();
_nResult := _fbDevice.GetLinkControlData();

AssertEquals(Expected := _nExpected,
             Actual := _nResult,
             Message := 'Value is not correct');	
TEST_FINISHED();

TEST('Get nStatus');
_nExpected := 255;
_fbDevice.SetStatus(_nExpected);
_fbDevice();
_nResult := _fbDevice.nStatus;

AssertEquals(Expected := _nExpected,
             Actual := _nResult,
             Message := 'Value is not correct');	
TEST_FINISHED();

TEST('Get nDataOut');
_nExpected := 255;
_fbDevice.SetLinkStatusData(_nExpected);
_fbDevice();
_nResult := _fbDevice.nStatusData;

AssertEquals(Expected := _nExpected,
             Actual := _nResult,
             Message := 'Value is not correct');	
TEST_FINISHED();

END_FUNCTION_BLOCK

// ---- Devices/Basic/FB_DeviceByte.TcPOU
(*
	Basic device with extended interface:
	nControl BYTE: From TwinCAT >>> To Unity
	nStatus BYTE: FROM Unity >>> TO TwinCAT	
	nControlData BYTE: From TwinCAT >>> To Unity
	nStatusData BYTE: FROM Unity >>> TO TwinCAT	
*)
FUNCTION_BLOCK FB_DeviceByte EXTENDS FB_LinkDataByte
VAR_INPUT		
	nControl  			: BYTE;
	nControlData  		: BYTE;
END_VAR

VAR_OUTPUT
	nStatus  			: BYTE;
	nStatusData  		: BYTE;
END_VAR

SUPER^();
Control := nControl;
ControlData := nControlData;
nStatus := Status;
nStatusData := StatusData;

END_FUNCTION_BLOCK

// ---- Tests/Devices/FB_DeviceWord_Test.TcPOU
FUNCTION_BLOCK FB_DeviceWord_Test EXTENDS TcUnit.FB_TestSuite
VAR
	_fbDevice 		: FB_DeviceWord;
	_nExpected 		: WORD;
	_nResult 		: WORD;
	_nValue 		: WORD := 16#FF;
END_VAR

TEST('Set nControl');
_nExpected := 255;
_fbDevice.nControl := 255;
_fbDevice();
_nResult := _fbDevice.GetControl();

AssertEquals(Expected := _nExpected,
             Actual := _nResult,
             Message := 'Value is not correct');	
TEST_FINISHED();

TEST('Set nDataIn');
_nExpected := _nValue;
_fbDevice.nControlData := _nExpected;
_fbDevice();
_nResult := _fbDevice.GetLinkControlData();

AssertEquals(Expected := _nExpected,
             Actual := _nResult,
             Message := 'Value is not correct');	
TEST_FINISHED();

TEST('Get nStatus');
_nExpected := 255;
_fbDevice.SetStatus(255);
_fbDevice();
_nResult := _fbDevice.nStatus;

AssertEquals(Expected := _nExpected,
             Actual := _nResult,
             Message := 'Value is not correct');	
TEST_FINISHED();

TEST('Get nDataOut');
_nExpected := _nValue;
_fbDevice.SetLinkStatusData(_nExpected);
_fbDevice();
_nResult := _fbDevice.nStatusData;

AssertEquals(Expected := _nExpected,
             Actual := _nResult,
             Message := 'Value is not correct');	
TEST_FINISHED();

END_FUNCTION_BLOCK

// ---- Devices/Basic/FB_DeviceWord.TcPOU
(*
	Basic device with extended interface:
	nControl BYTE: From TwinCAT >>> To Unity
	nStatus BYTE: FROM Unity >>> TO TwinCAT	
	nControlData WORD: From TwinCAT >>> To Unity
	nStatusData WORD: FROM Unity >>> TO TwinCAT	
*)
FUNCTION_BLOCK FB_DeviceWord EXTENDS FB_LinkDataWord
VAR_INPUT		
	nControl  			: BYTE;
	nControlData  		: WORD;
END_VAR

VAR_OUTPUT
	nStatus  			: BYTE;
	nStatusData  		: WORD;
END_VAR

SUPER^();
Control := nControl;
ControlData := nControlData;
nStatus := Status;
nStatusData := StatusData;

END_FUNCTION_BLOCK

// ---- Common/Links/FB_LinkDataWord.TcPOU
(*
	Link component with additional interface:
	Control BYTE: From TwinCAT >>> To Unity	(Default)
	Status BYTE: FROM Unity >>> TO TwinCAT	(Default)
	ControlData WORD: From TwinCAT >>> To Unity		
	StatusData WORD: FROM Unity >>> TO TwinCAT		
*)
FUNCTION_BLOCK FB_LinkDataWord EXTENDS FB_LinkDevice
VAR	
	{attribute 'simulation_interface'}
	ControlData		AT %Q* : WORD;
	{attribute 'simulation_interface'}
	StatusData		AT %I* : WORD;	
END_VAR

SUPER^();

METHOD INTERNAL GetLinkControlData : WORD
GetLinkControlData := ControlData;
END_METHOD

METHOD INTERNAL SetLinkStatusData : BOOL
VAR_INPUT
	nStatusData : WORD;
END_VAR
StatusData := nStatusData;
END_METHOD

END_FUNCTION_BLOCK

// ---- Tests/Devices/FB_DeviceDWord_Test.TcPOU
FUNCTION_BLOCK FB_DeviceDWord_Test EXTENDS TcUnit.FB_TestSuite
VAR
	_fbDevice 		: FB_DeviceDWord;
	_nExpected 		: DWORD;
	_nResult 		: DWORD;
	_nValue 		: DWORD := 16#FFAA;
END_VAR

TEST('Set nControl');
_nExpected := 255;
_fbDevice.nControl := 255;
_fbDevice();
_nResult := _fbDevice.GetControl();

AssertEquals(Expected := _nExpected,
             Actual := _nResult,
             Message := 'Value is not correct');	
TEST_FINISHED();

TEST('Set nDataIn');
_nExpected := _nValue;
_fbDevice.nControlData := _nExpected;
_fbDevice();
_nResult := _fbDevice.GetLinkControlData();

AssertEquals(Expected := _nExpected,
             Actual := _nResult,
             Message := 'Value is not correct');	
TEST_FINISHED();

TEST('Get nStatus');
_nExpected := 255;
_fbDevice.SetStatus(255);
_fbDevice();
_nResult := _fbDevice.nStatus;

AssertEquals(Expected := _nExpected,
             Actual := _nResult,
             Message := 'Value is not correct');	
TEST_FINISHED();

TEST('Get nDataOut');
_nExpected := _nValue;
_fbDevice.SetLinkStatusData(_nExpected);
_fbDevice();
_nResult := _fbDevice.nStatusData;

AssertEquals(Expected := _nExpected,
             Actual := _nResult,
             Message := 'Value is not correct');	
TEST_FINISHED();

END_FUNCTION_BLOCK

// ---- Devices/Basic/FB_DeviceDWord.TcPOU
(*
	Basic device with extended interface:
	nControl BYTE: From TwinCAT >>> To Unity
	nStatus BYTE: FROM Unity >>> TO TwinCAT	
	nControlData DWORD: From TwinCAT >>> To Unity
	nStatusData DWORD: FROM Unity >>> TO TwinCAT	
*)
FUNCTION_BLOCK FB_DeviceDWord EXTENDS FB_LinkDataDWord
VAR_INPUT		
	nControl  			: BYTE;
	nControlData 		: DWORD;
END_VAR

VAR_OUTPUT
	nStatus  			: BYTE;
	nStatusData  		: DWORD;
END_VAR

SUPER^();
Control := nControl;
ControlData := nControlData;
nStatus := Status;
nStatusData := StatusData;

END_FUNCTION_BLOCK

// ---- Tests/Devices/FB_DeviceLWord_Test.TcPOU
FUNCTION_BLOCK FB_DeviceLWord_Test EXTENDS TcUnit.FB_TestSuite
VAR
	_fbDevice 		: FB_DeviceLWord;
	_nExpected 		: LWORD;
	_nResult 		: LWORD;
	_nValue 		: LWORD := 16#FFAABBCC;
END_VAR

TEST('Set nControl');
_nExpected := 255;
_fbDevice.nControl := 255;
_fbDevice();
_nResult := _fbDevice.GetControl();

AssertEquals(Expected := _nExpected,
             Actual := _nResult,
             Message := 'Value is not correct');	
TEST_FINISHED();

TEST('Set nDataIn');
_nExpected := _nValue;
_fbDevice.nControlData := _nExpected;
_fbDevice();
_nResult := _fbDevice.GetLinkControlData();

AssertEquals(Expected := _nExpected,
             Actual := _nResult,
             Message := 'Value is not correct');	
TEST_FINISHED();

TEST('Get nStatus');
_nExpected := 255;
_fbDevice.SetStatus(255);
_fbDevice();
_nResult := _fbDevice.nStatus;

AssertEquals(Expected := _nExpected,
             Actual := _nResult,
             Message := 'Value is not correct');	
TEST_FINISHED();

TEST('Get nDataOut');
_nExpected := _nValue;
_fbDevice.SetLinkStatusData(_nExpected);
_fbDevice();
_nResult := _fbDevice.nStatusData;

AssertEquals(Expected := _nExpected,
             Actual := _nResult,
             Message := 'Value is not correct');	
TEST_FINISHED();

END_FUNCTION_BLOCK

// ---- Devices/Basic/FB_DeviceLWord.TcPOU
(*
	Basic device with extended interface:
	nControl BYTE: From TwinCAT >>> To Unity
	nStatus BYTE: FROM Unity >>> TO TwinCAT	
	nControlData LWORD: From TwinCAT >>> To Unity
	nStatusData LWORD: FROM Unity >>> TO TwinCAT	
*)
FUNCTION_BLOCK FB_DeviceLWord EXTENDS FB_LinkDataLWord
VAR_INPUT		
	nControl  			: BYTE;
	nControlData  		: LWORD;
END_VAR

VAR_OUTPUT
	nStatus  			: BYTE;
	nStatusData  		: LWORD;
END_VAR

SUPER^();
Control := nControl;
ControlData := nControlData;
nStatus := Status;
nStatusData := StatusData;

END_FUNCTION_BLOCK

// ---- Common/Links/FB_LinkDataLWord.TcPOU
(*
	Link component with additional interface:
	Control BYTE: From TwinCAT >>> To Unity	(Default)
	Status BYTE: FROM Unity >>> TO TwinCAT	(Default)
	ControlData LWORD: From TwinCAT >>> To Unity		
	StatusData LWORD: FROM Unity >>> TO TwinCAT		
*)
FUNCTION_BLOCK FB_LinkDataLWord EXTENDS FB_LinkDevice
VAR	
	{attribute 'simulation_interface'}
	ControlData		AT %Q* : LWORD;
	{attribute 'simulation_interface'}
	StatusData		AT %I* : LWORD;
END_VAR

SUPER^();

METHOD INTERNAL GetLinkControlData : LWORD
GetLinkControlData := ControlData;
END_METHOD

METHOD INTERNAL SetLinkStatusData : BOOL
VAR_INPUT
	nStatusData : LWORD;
END_VAR
StatusData := nStatusData;
END_METHOD

END_FUNCTION_BLOCK

// ---- Tests/Devices/FB_DeviceReal_Test.TcPOU
FUNCTION_BLOCK FB_DeviceReal_Test EXTENDS TcUnit.FB_TestSuite
VAR
	_fbDevice 		: FB_DeviceReal;
	_fExpected 		: REAL;
	_fResult 		: REAL;
	_fValue 		: REAL := 16#FF;
END_VAR

TEST('Set nControl');
_fExpected := 255;
_fbDevice.nControl := 255;
_fbDevice();
_fResult := _fbDevice.GetControl();

AssertEquals(Expected := _fExpected,
             Actual := _fResult,
             Message := 'Value is not correct');	
TEST_FINISHED();

TEST('Set nDataIn_1');
_fExpected := 1000;
_fbDevice.fControlData := _fExpected;
_fbDevice();
_fResult := _fbDevice.GetLinkControlData();

AssertEquals(Expected := _fExpected,
             Actual := _fResult,
             Message := 'Value is not correct');	
TEST_FINISHED();

TEST('Set nDataIn_2');
_fExpected := -1000;
_fbDevice.fControlData := _fExpected;
_fbDevice();
_fResult := _fbDevice.GetLinkControlData();

AssertEquals(Expected := _fExpected,
             Actual := _fResult,
             Message := 'Value is not correct');	
TEST_FINISHED();

TEST('Get nStatus');
_fExpected := 255;
_fbDevice.SetStatus(255);
_fbDevice();
_fResult := _fbDevice.nStatus;

AssertEquals(Expected := _fExpected,
             Actual := _fResult,
             Message := 'Value is not correct');	
TEST_FINISHED();

TEST('Get nDataOut_1');
_fExpected := 1000;
_fbDevice.SetLinkStatusData(_fExpected);
_fbDevice();
_fResult := _fbDevice.fStatusData;

AssertEquals(Expected := _fExpected,
             Actual := _fResult,
             Message := 'Value is not correct');	
TEST_FINISHED();

TEST('Get nDataOut_2');
_fExpected := -1000;
_fbDevice.SetLinkStatusData(_fExpected);
_fbDevice();
_fResult := _fbDevice.fStatusData;

AssertEquals(Expected := _fExpected,
             Actual := _fResult,
             Message := 'Value is not correct');	
TEST_FINISHED();

END_FUNCTION_BLOCK

